DATA_BLOCK "DB7300_INTERLOCK_GENERAL"   // DB7300
{ S7_Optimized_Access := 'FALSE'; DB_Accessible_From_OPC_UA := 'FALSE' }
AUTHOR : ETXETAR
VERSION : 1.0
// stored: AutoNumber false, DBAccessibleFromOPCUA false, DBAccessibleFromWebserver true, IsOnlyStoredInLoadMemory false, IsWriteProtectedInAS false
   VAR RETAIN
      GENERAL_MACHINE : Struct
         FROM_CELL_TO_MACHINE_GENERAL : Struct
            MEAS_STA_START_CYCLE : Bool;   // CELL MEASURING STATION START CYCLE
            MEAS_STA_CALIB_CYCLE : Bool;   // CELL MEASURING STATION CALIBRATION CYCLE
            MEAS_STA_HOME_REQ : Bool;   // CELL MEASURING STATION HOME REQUEST
            MEAS_STA_FAULT : Bool;   // CELL MEASURING STATION FAULT
            MEAS_STA_RESET : Bool;   // CELL MEASURING STATION RESET
            MEAS_STA_ROBOT_OUT_OF_COLLISION : Bool;
            MEAS_STA_PART_LOADED : Bool;   // CELL MEASURING STATION PART LOADED
            MEAS_STA_PART_UNLOADED : Bool;   // CELL MEASURING STATION PART UNLOADED
            MEAS_STA_SEQ_RUNNING : Bool;   // CELL MEASURING STATION SEQUENCE RUNNING
            CELL_COOLING_DEGRADED_MODE : Bool;   // CELL COOLING DEGRADED MODE
            CELL_STARVED : Bool;   // CELL STARVED
            CELL_BLOCKED : Bool;   // CELL BLOCKED
            CELL_LOADING_ACTIVE : Bool;   // CELL LOADING ACTIVE
            CELL_CALIBRATION_CYCLE_REQUIRED : Bool;   // CELL CALIBRATION CYCLE REQUIRED
         END_STRUCT;
         FROM_ROBOT_TO_UNIT_1 : Struct
            HEARTBEAT : Bool;   // ROBOT HEARTBEAT
            EMERG_STOP_OK : Bool;   // ROBOT EMERGENCY STOP OK
            ROBOT_FAULT : Bool;   // ROBOT FAULT
            SAFETY_DOOR_CLSD_LOCKD : Bool;   // ROBOT SAFETY DOOR CLOSED AND LOCKED
            CELL_EMPTY : Bool;   // ROBOT CELL EMPTY
            IN_SEMIAUTO_MODE : Bool;   // ROBOT SEMIAUTO MODE SELECTED
            IN_MANUAL_MODE : Bool;   // ROBOT MANUAL MODE SELECTED
            IN_AUTO_MODE : Bool;   // ROBOT AUTO MODE SELECTED
            IN_AUTO_CYCLE_RUN : Bool;   // ROBOT CYCLE RUNNING IN AUTOMATIC MODE
            RUN_OUT_REQUEST : Bool;   // ROBOT MACHINE RUN OUT REQUEST
            RUN_OUT_COMPLETED : Bool;   // ROBOT RUN OUT COMPLETED
            SAFETY_DOOR_OPEN_REQ : Bool;   // ROBOT ANY CELL SAFETY DOOR OPEN REQUEST
            OK_TO_OPEN_SAFETY_GATES : Bool;   // ROBOT OK TO OPEN SAFETY GATES
            READY_TO_SERVICE : Bool;   // ROBOT READY TO SERVICE MACHINE
            OUT_OF_COLLISION_MACHINE : Bool;   // ROBOT OUT OF COLLISION MACHINE
            OUT_OF_COLLISION_FIXTURE : Bool;   // ROBOT OUT OF COLLISION FIXTURE
            PART_ENABLED : Bool;   // ROBOT PART ENABLED
            PART_FACE_R_TO_DELIVER : Bool;   // ROBOT PART FACE R TO DELIVER IMMEDIATELY
            PART_FACE_N_TO_DELIVER : Bool;   // ROBOT PART FACE N TO DELIVER IMMEDIATELY
            OUT_OF_PARTS_FACE_R_TO_DELIVER : Bool;   // ROBOT OUT OF PARTS FACE R IN CELL TO DELIVER
            OUT_OF_PARTS_FACE_N_TO_DELIVER : Bool;   // ROBOT OUT OF PARTS FACE N IN CELL TO DELIVER
            PART_LOADED : Bool;   // ROBOT PART LOADED
            PART_UNLOADED : Bool;   // ROBOT PART UNLOADED
            FIX_SKIP_REQ : Bool;   // ROBOT FIXTURE SKIP REQUEST
            PART_TYPE_CHANGE_REQ : Bool;   // ROBOT PART TYPE CHANGE REQUEST
            PART_TYPE : Byte;   // ROBOT PART TYPE
         END_STRUCT;
         FROM_ROBOT_TO_UNIT_2 : Struct
            HEARTBEAT : Bool;   // ROBOT HEARTBEAT
            EMERG_STOP_OK : Bool;   // ROBOT EMERGENCY STOP OK
            ROBOT_FAULT : Bool;   // ROBOT FAULT
            SAFETY_DOOR_CLSD_LOCKD : Bool;   // ROBOT SAFETY DOOR CLOSED AND LOCKED
            CELL_EMPTY : Bool;   // ROBOT CELL EMPTY
            IN_SEMIAUTO_MODE : Bool;   // ROBOT SEMIAUTO MODE SELECTED
            IN_MANUAL_MODE : Bool;   // ROBOT MANUAL MODE SELECTED
            IN_AUTO_MODE : Bool;   // ROBOT AUTO MODE SELECTED
            IN_AUTO_CYCLE_RUN : Bool;   // ROBOT CYCLE RUNNING IN AUTOMATIC MODE
            RUN_OUT_REQUEST : Bool;   // ROBOT MACHINE RUN OUT REQUEST
            RUN_OUT_COMPLETED : Bool;   // ROBOT RUN OUT COMPLETED
            SAFETY_DOOR_OPEN_REQ : Bool;   // ROBOT ANY CELL SAFETY DOOR OPEN REQUEST
            OK_TO_OPEN_SAFETY_GATES : Bool;   // ROBOT OK TO OPEN SAFETY GATES
            READY_TO_SERVICE : Bool;   // ROBOT READY TO SERVICE MACHINE
            OUT_OF_COLLISION_MACHINE : Bool;   // ROBOT OUT OF COLLISION MACHINE
            OUT_OF_COLLISION_FIXTURE : Bool;   // ROBOT OUT OF COLLISION FIXTURE
            PART_ENABLED : Bool;   // ROBOT PART ENABLED
            PART_FACE_R_TO_DELIVER : Bool;   // ROBOT PART FACE R TO DELIVER IMMEDIATELY
            PART_FACE_N_TO_DELIVER : Bool;   // ROBOT PART FACE N TO DELIVER IMMEDIATELY
            OUT_OF_PARTS_FACE_R_TO_DELIVER : Bool;   // ROBOT OUT OF PARTS FACE R IN CELL TO DELIVER
            OUT_OF_PARTS_FACE_N_TO_DELIVER : Bool;   // ROBOT OUT OF PARTS FACE N IN CELL TO DELIVER
            PART_LOADED : Bool;   // ROBOT PART LOADED
            PART_UNLOADED : Bool;   // ROBOT PART UNLOADED
            FIX_SKIP_REQ : Bool;   // ROBOT FIXTURE SKIP REQUEST
            PART_TYPE_CHANGE_REQ : Bool;   // ROBOT PART TYPE CHANGE REQUEST
            PART_TYPE : Byte;   // ROBOT PART TYPE
         END_STRUCT;
      END_STRUCT;
      POWDER_PLC : Struct
         GENERAL : Struct
            LIFE_BIT : Bool;   // LIFE BIT
            SELECTED_ARGON_GAS : Bool;   // SELECTED ARGON GAS
            SELECTED_NITROGEN_GAS : Bool;   // SELECTED NITROGEN GAS
            SELECTED_IMPERIAL_SYSTEM : Bool;   // SELECTED IMPERIAL SYSTEM
            SELECTED_METRIC_SYSTEM : Bool;   // SELECTED METRIC SYSTEM
            POWDER_PLC_AUTO_MODE : Bool;   // POWDER PLC IN AUTO MODE
            POWDER_PLC_MAN_MODE : Bool;   // POWDER PLC IN MANUAL MODE
         END_STRUCT;
         FROM_POWDER_TO_UNIT_1 : Struct
            POWDER_UNIT_1_READY_TO_RUN : Bool;   // POWDER UNIT 1 READY TO RUN
            POWDER_UNIT_1_STOPPED : Bool;   // POWDER UNIT 1 STOPPED
            SWITCHED_ON_POWDER_UNIT_1 : Bool;   // SWITCHED ON POWDER UNIT 1
            SWITCHED_OFF_POWDER_UNIT_1 : Bool;   // SWITCHED OFF POWDER UNIT 1
            SWITCHED_ON_TEMPERATURE_JACKET_UNIT_1 : Bool;   // SWITCHED ON TEMPERATURE JACKET UNIT 1
            SWITCHED_OFF_TEMPERATURE_JACKET_UNIT_1 : Bool;   // SWITCHED OFF TEMPERATURE JACKET UNIT 1
            U1_PF_1_LINE_1_LOW_POWDER : Bool;   // UNIT 1 POWDER FEEDER 1 LINE 1 LOW POWDER LEVEL
            U1_PF_1_LINE_2_LOW_POWDER : Bool;   // UNIT 1 POWDER FEEDER 1 LINE 2 LOW POWDER LEVEL
            POWDER_UNIT_1_ALARM : Bool;   // POWDER UNIT 1 ALARM
            UNIT_1_POWDER_FEEDER_1_CARRIER_GAS_ACTUAL_LINE_1 : Real;   // UNIT 1 POWDER FEEDER 1 CARRIER GAS ACTUAL LINE 1
            UNIT_1_POWDER_FEEDER_1_DISK_SPEED_ACTUAL_LINE_1 : Real;   // UNIT 1 POWDER FEEDER 1 DISK SPEED ACTUAL LINE 1
            UNIT_1_POWDER_FEEDER_1_STIRRER_SPEED_ACTUAL_LINE_1 : Real;   // UNIT 1 POWDER FEEDER 1 STIRRER SPEED ACTUAL LINE 1
            UNIT_1_POWDER_FEEDER_1_HOPPER_TEMPERATURE_ACTUAL_LINE_1 : Real;   // UNIT 1 POWDER FEEDER 1 HOPPER TEMPERATURE ACTUAL LINE 1
            UNIT_1_POWDER_FEEDER_1_CARRIER_GAS_ACTUAL_LINE_2 : Real;   // UNIT 1 POWDER FEEDER 1 CARRIER GAS ACTUAL LINE 2
            UNIT_1_POWDER_FEEDER_1_DISK_SPEED_ACTUAL_LINE_2 : Real;   // UNIT 1 POWDER FEEDER 1 DISK SPEED ACTUAL LINE 2
            UNIT_1_POWDER_FEEDER_1_STIRRER_SPEED_ACTUAL_LINE_2 : Real;   // UNIT 1 POWDER FEEDER 1 STIRRER SPEED ACTUAL LINE 2
            UNIT_1_POWDER_FEEDER_1_HOPPER_TEMPERATURE_ACTUAL_LINE_2 : Real;   // UNIT 1 POWDER FEEDER 1 HOPPER TEMPERATURE ACTUAL LINE 2
         END_STRUCT;
         FROM_POWDER_TO_UNIT_2 : Struct
            POWDER_UNIT_2_READY_TO_RUN : Bool;   // POWDER UNIT 2 READY TO RUN
            POWDER_UNIT_2_STOPPED : Bool;   // POWDER UNIT 2 STOPPED
            SWITCHED_ON_POWDER_UNIT_2 : Bool;   // SWITCHED ON POWDER UNIT 2
            SWITCHED_OFF_POWDER_UNIT_2 : Bool;   // SWITCHED OFF POWDER UNIT 2
            SWITCHED__ON_TEMPERATURE_JACKET_UNIT_2 : Bool;   // SWITCHED ON TEMPERATURE JACKET UNIT 2
            SWITCHED_OFF_TEMPERATURE_JACKET_UNIT_2 : Bool;   // SWITCHED OFF TEMPERATURE JACKET UNIT 2
            U2_PF_1_LINE_1_LOW_POWDER : Bool;   // UNIT 2 POWDER FEEDER 1 LINE 1 LOW POWDER LEVEL
            U2_PF_1_LINE_2_LOW_POWDER : Bool;   // UNIT 2 POWDER FEEDER 1 LINE 2 LOW POWDER LEVEL
            U2_PF_2_LINE_2_LOW_POWDER : Bool;   // UNIT 2 POWDER FEEDER 2 LINE 2 LOW POWDER LEVEL
            POWDER_UNIT_2_ALARM : Bool;   // POWDER UNIT 2 ALARM
            UNIT_2_POWDER_FEEDER_1_CARRIER_GAS_ACTUAL_LINE_1 : Real;   // UNIT 2 POWDER FEEDER 1 CARRIER GAS ACTUAL LINE 1
            UNIT_2_POWDER_FEEDER_1_CARRIER_GAS_ACTUAL_LINE_2 : Real;   // UNIT 2 POWDER FEEDER 1 CARRIER GAS ACTUAL LINE 2
            UNIT_2_POWDER_FEEDER_1_DISK_SPEED_ACTUAL_LINE_1 : Real;   // UNIT 2 POWDER FEEDER 1 DISK SPEED ACTUAL LINE 1
            UNIT_2_POWDER_FEEDER_1_DISK_SPEED_ACTUAL_LINE_2 : Real;   // UNIT 2 POWDER FEEDER 1 DISK SPEED ACTUAL LINE 2
            UNIT_2_POWDER_FEEDER_1_STIRRER_SPEED_ACTUAL_LINE_1 : Real;   // UNIT 2 POWDER FEEDER 1 STIRRER SPEED ACTUAL LINE 1
            UNIT_2_POWDER_FEEDER_1_STIRRER_SPEED_ACTUAL_LINE_2 : Real;   // UNIT 2 POWDER FEEDER 1 STIRRER SPEED ACTUAL LINE 2
            UNIT_2_POWDER_FEEDER_1_HOPPER_TEMPERATURE_ACTUAL_LINE_1 : Real;   // UNIT 2 POWDER FEEDER 1 HOPPER TEMPERATURE ACTUAL LINE 1
            UNIT_2_POWDER_FEEDER_1_HOPPER_TEMPERATURE_ACTUAL_LINE_2 : Real;   // UNIT 2 POWDER FEEDER 1 HOPPER TEMPERATURE ACTUAL LINE 2
            UNIT_2_POWDER_FEEDER_2_CARRIER_GAS_ACTUAL_LINE_1 : Real;   // UNIT 2 POWDER FEEDER 2 CARRIER GAS ACTUAL LINE 1
            UNIT_2_POWDER_FEEDER_2_CARRIER_GAS_ACTUAL_LINE_2 : Real;   // UNIT 2 POWDER FEEDER 2 CARRIER GAS ACTUAL LINE 2
            UNIT_2_POWDER_FEEDER_2_DISK_SPEED_ACTUAL_LINE_1 : Real;   // UNIT 2 POWDER FEEDER 2 DISK SPEED ACTUAL LINE 1
            UNIT_2_POWDER_FEEDER_2_STIRRER_SPEED_ACTUAL_LINE_1 : Real;   // UNIT 2 POWDER FEEDER 2 STIRRER SPEED ACTUAL LINE 1
            UNIT_2_POWDER_FEEDER_2_DISK_SPEED_ACTUAL_LINE_2 : Real;   // UNIT 2 POWDER FEEDER 2 DISK SPEED ACTUAL LINE 2
            UNIT_2_POWDER_FEEDER_2_STIRRER_SPEED_ACTUAL_LINE_2 : Real;   // UNIT 2 POWDER FEEDER 2 STIRRER SPEED ACTUAL LINE 2
            UNIT_2_POWDER_FEEDER_2_HOPPER_TEMPERATURE_ACTUAL_LINE_1 : Real;   // UNIT 2 POWDER FEEDER 2 HOPPER TEMPERATURE ACTUAL LINE 1
            UNIT_2_POWDER_FEEDER_2_HOPPER_TEMPERATURE_ACTUAL_LINE_2 : Real;   // UNIT 2 POWDER FEEDER 2 HOPPER TEMPERATURE ACTUAL LINE 2
         END_STRUCT;
      END_STRUCT;
      LOAD_UNLOAD : Struct
         UNIT_1 : "LOAD_UNLOAD_ETXETAR_ROBOT_CELL";
         UNIT_2 : "LOAD_UNLOAD_ETXETAR_ROBOT_CELL";
         UNIT_3 : "LOAD_UNLOAD_ETXETAR_ROBOT_CELL";
      END_STRUCT;
      AUX_SIGNALS_INTERFACE : Struct
         GENERAL : Struct
            "MEASURING STATION FAULT" : Bool;   // CELL MEASURING STATION FAULT
            "DEGRADED MODE FAULT" : Bool;   // CELL COOLING DEGRADED MODE FAULT
            TIMER_MEASURING_IN_PRCS : TOF_TIME;   // TIMER MEASURING IN PROCESS
            TIMER_MEASURING_DONE : TOF_TIME;   // TIMER MEASURING DONE
         END_STRUCT;
         UNIT_1 : Struct
            LIFE_BIT_FAULT : Bool;   // HEARTBEAT COMMUNICATION ALARM
            EMERGENCY_STOP_ACTIVE : Bool;   // EMERGENCY STOP ACTIVE ALARM
            ROBOT_FAULT_INSIDE_OF_MACHINE : Bool;   // ROBOT FAULT ALARM INSIDE OF MACHINE
            ROBOT_FAULT_OUTSIDE_OF_MACHINE : Bool;   // ROBOT FAULT ALARM OUTSIDE OF MACHINE
            FACE_R_LOAD_REQ_AUX : Bool;   // FACE R LOAD REQUEST AUX
            FACE_N_LOAD_REQ_AUX : Bool;   // FACE N LOAD REQUEST AUX
            "LIFE SING COUNTER" : CTU_INT;
         END_STRUCT;
         UNIT_2 : Struct
            LIFE_BIT_FAULT : Bool;   // HEARTBEAT COMMUNICATION ALARM
            EMERGENCY_STOP_ACTIVE : Bool;   // EMERGENCY STOP ACTIVE ALARM
            ROBOT_FAULT_INSIDE_OF_MACHINE : Bool;   // ROBOT FAULT ALARM INSIDE OF MACHINE
            ROBOT_FAULT_OUTSIDE_OF_MACHINE : Bool;   // ROBOT FAULT ALARM OUTSIDE OF MACHINE
            FACE_R_LOAD_REQ_AUX : Bool;   // FACE R LOAD REQUEST AUX
            FACE_N_LOAD_REQ_AUX : Bool;   // FACE N LOAD REQUEST AUX
            "LIFE SING COUNTER" : CTU_INT;
         END_STRUCT;
         POWDER_PLC : Struct
            LIFE_BIT_FAULT : Bool;   // HEARTBEAT COMMUNICATION ALARM
            "LIFE SING COUNTER" : CTU_INT;
         END_STRUCT;
         AUX_0 : Bool;   // AUXILIARY 0
         AUX_1 : Bool;   // AUXILIARY 1
         AUX_2 : Bool;   // AUXILIARY 2
         AUX_3 : Bool;   // AUXILIARY 3
         AUX_4 : Bool;   // AUXILIARY 4
         AUX_5 : Bool;   // AUXILIARY 5
         AUX_6 : Bool;   // AUXILIARY 6
         AUX_7 : Bool;   // AUXILIARY 7
         AUX_8 : Bool;   // AUXILIARY 8
         AUX_9 : Bool;   // AUXILIARY 9
         AUX_10 : Bool;   // AUXILIARY 10
         AUX_11 : Bool;   // AUXILIARY 11
         AUX_12 : Bool;   // AUXILIARY 12
         AUX_13 : Bool;   // AUXILIARY 13
         AUX_14 : Bool;   // AUXILIARY 14
         AUX_15 : Bool;   // AUXILIARY 15
         TIMER_IS_SEOC_ROBOT_FAULT_UNIT_1 : TON_TIME;   // TIMER IS SEOC ROBOT FAULT UNIT 1
         TIMER_IS_SEOC_ROBOT_FAULT_UNIT_2 : TON_TIME;   // TIMER IS SEOC ROBOT FAULT UNIT 2
         TIMER_SEOC_ROBOT_FAULT_UNIT_1 : TON_TIME;   // TIMER SEOC ROBOT FAULT UNIT 1
         TIMER_SEOC_ROBOT_FAULT_UNIT_2 : TON_TIME;   // TIMER SEOC ROBOT FAULT UNIT 2
      END_STRUCT;
      PART_A : Struct
         UNIT_1 : "PART_STATUS_CLADDING";
         UNIT_2 : "PART_STATUS_CLADDING";
         UNIT_3 : "PART_STATUS_CLADDING";
      END_STRUCT;
   END_VAR
BEGIN
   AUX_SIGNALS_INTERFACE.GENERAL.TIMER_MEASURING_IN_PRCS.PT := T#3s;
   AUX_SIGNALS_INTERFACE.GENERAL.TIMER_MEASURING_DONE.PT := T#3s;
   AUX_SIGNALS_INTERFACE.TIMER_IS_SEOC_ROBOT_FAULT_UNIT_1.PT := T#2M;
   AUX_SIGNALS_INTERFACE.TIMER_IS_SEOC_ROBOT_FAULT_UNIT_2.PT := T#2M;
   AUX_SIGNALS_INTERFACE.TIMER_SEOC_ROBOT_FAULT_UNIT_1.PT := T#2M;
   AUX_SIGNALS_INTERFACE.TIMER_SEOC_ROBOT_FAULT_UNIT_2.PT := T#2M;
END_DATA_BLOCK

DATA_BLOCK "DB7400_QUALITY"   // DB7400
{ S7_Optimized_Access := 'FALSE'; DB_Accessible_From_OPC_UA := 'FALSE' }
AUTHOR : ETXETAR
VERSION : 1.0
// stored: AutoNumber false, DBAccessibleFromOPCUA false, DBAccessibleFromWebserver true, IsOnlyStoredInLoadMemory false, IsWriteProtectedInAS false
   VAR RETAIN
      OPTIONS : Struct   // OPTIONS
         QC_STOP_END_OF_CYCLE : Bool;   // QC STOP END OF CYCLE
         SP11_WORKS_TWO_PARTS : Bool;   // SP11 WORKS TWO PARTS
         SP12_WORKS_TWO_PARTS : Bool;   // SP12 WORKS TWO PARTS
         SP21_WORKS_TWO_PARTS : Bool;   // SP21 WORKS TWO PARTS
         SP22_WORKS_TWO_PARTS : Bool;   // SP22 WORKS TWO PARTS
         FIRST_SCAN : Bool;   // FIRST SCAN
         CYCLE_INTERRUPTED : Bool;   // CYCLE INTERRUPTED
         ANY_TOOL_NEW : Bool;   // ANY TOOL NEW
         BROKEN_TOOL : Bool;   // BROKEN TOOL
         ALL_BROKEN_TOOL : Bool;   // ALL BROKEN TOOL IF ONE TOOL IS BROKEN ALL PARTS ARE MARKED
         ONE_COUNTER : Bool;   // ONE COUNTER
         COUNTER_PER_PART : Bool;   // COUNTER PER PART
         CMM_QUALITY_CHECK : Bool;   // CMM QUALITY CHECK
         SURFACE_QUALITY_CHECK : Bool;   // SURFACE QUALITY CHECK
      END_STRUCT;
      PART_CONTROL : Struct   // PART CONTROL
         HMI_QUALITY_HALF_PART : Bool;   // HMI QUALITY HALF PART
         HMI_QUALITY_FULL_PART : Bool;   // HMI QUALITY FULL PART
         HMI_QUALITY_CANCEL : Bool;   // HMI QUALITY CANCEL
         HMI_QUALITY_NOK : Bool;   // HMI QUALITY NOK
         HMI_QUALITY_OK : Bool;   // HMI QUALITY OK
         HALF_QUALITY_PART_SELECTED : Bool;   // HALF QUALITY PART SELECTED
         FULL_QUALITY_PART_SELECTED : Bool;   // FULL QUALITY PART SELECTED
         PART_QUALITY_ON_DEMAND : Bool;   // PART QUALITY ON DEMAND
         QUALITY_AUX_WARNING : Bool;   // QUALITY AUX WARNING
         QUALITY_AUX_FAULT : Bool;   // QUALITY AUX FAULT
         QUALITY_PART : Bool;   // QUALITY PART
         FIXTURE_2_QUALITY : Bool;   // FIXTURE 2 QUALITY
         U01_FIXTURE_1_PART_P : Bool;   // UNIT 01 FIXTURE 1 PART A PULSE
         U01_FIXTURE_2_PART_P : Bool;   // UNIT 01 FIXTURE 2 PART A PULSE
         U01_FIXTURE_3_PART_P : Bool;   // UNIT 01 FIXTURE 3 PART A PULSE
         U01_FIXTURE_4_PART_P : Bool;   // UNIT 01 FIXTURE 4 PART A PULSE
         U02_FIXTURE_1_PART_P : Bool;   // UNIT 02 FIXTURE 1 PART A PULSE
         U02_FIXTURE_2_PART_P : Bool;   // UNIT 02 FIXTURE 2 PART A PULSE
         U02_FIXTURE_3_PART_P : Bool;   // UNIT 02 FIXTURE 3 PART A PULSE
         U02_FIXTURE_4_PART_P : Bool;   // UNIT 02 FIXTURE 4 PART A PULSE
         U01_FIXTURE_1_PART_DEMAND : Bool;   // UNIT 01 FIXTURE 1 PART A DEMAND
         U01_FIXTURE_2_PART_DEMAND : Bool;   // UNIT 01 FIXTURE 2 PART A DEMAND
         U01_FIXTURE_3_PART_DEMAND : Bool;   // UNIT 01 FIXTURE 3 PART A DEMAND
         U01_FIXTURE_4_PART_DEMAND : Bool;   // UNIT 01 FIXTURE 4 PART A DEMAND
         U02_FIXTURE_1_PART_DEMAND : Bool;   // UNIT 02 FIXTURE 1 PART A DEMAND
         U02_FIXTURE_2_PART_DEMAND : Bool;   // UNIT 02 FIXTURE 2 PART A DEMAND
         U02_FIXTURE_3_PART_DEMAND : Bool;   // UNIT 02 FIXTURE 3 PART A DEMAND
         U02_FIXTURE_4_PART_DEMAND : Bool;   // UNIT 02 FIXTURE 4 PART A DEMAND
         PART_NOK : Bool;   // PART QUALITY DEMAND NOK ALARM
      END_STRUCT;
      PART_TYPE : Struct   // PART TYPE
         PART_TYPE_CHANGE_AUX : Bool;   // PART TYPE CHANGE AUXILIARY
         FIXTURE_1_PART_TYPE_CHANGE : Bool;   // FIXTURE 1 PART TYPE CHANGE
         FIXTURE_2_PART_TYPE_CHANGE : Bool;   // FIXTURE 2 PART TYPE CHANGE
         FIXTURE_3_PART_TYPE_CHANGE : Bool;   // FIXTURE 3 PART TYPE CHANGE
         FIXTURE_4_PART_TYPE_CHANGE : Bool;   // FIXTURE 4 PART TYPE CHANGE
         QUALITY_PART_TYPE_CHANGE : Bool;   // QUALITY AFTER PART TYPE CHANGE
         QUALITY_PART_NOK : Bool;   // QUALITY PART AFTER PART TYPE CHANGE NOK ALARM
      END_STRUCT;
      FIRST_CYCLE : Struct   // FIRST CYCLE
         FIRST_SCAN_AUX : Bool;   // FIRST SCAN AUXILIARY
         QUALITY_FIRST_CYCLE : Bool;   // QUALITY FIRST CYCLE
         FIXTURE_2_FIRST_CYCLE : Bool;   // FIXTURE 2 FIRST CYCLE
         FIXTURE_1_PART_A : Bool;   // FIXTURE 1 PART A FIRST CYCLE
         FIXTURE_1_PART_A_NOK : Bool;   // FIXTURE 1 PART A FIRST CYCLE NOK ALARM
      END_STRUCT;
      CYCLE_INTERRUPTED : Struct   // CYCLE INTERRUPTED
         CYCLE_INTERRUPTED_AUX : Bool;   // CYCLE INTERRUPTED AUXILIARY
         CYCLE_INTERRUPTED_AUX_P : Bool;   // CYCLE INTERRUPTED AUXILIARY PULSE
         FIXTURE_1_CYCLE_INTERRUPTED : Bool;   // FIXTURE 1 CYCLE INTERRUPTED
         FIXTURE_2_CYCLE_INTERRUPTED : Bool;   // FIXTURE 2 CYCLE INTERRUPTED
         FIXTURE_1_PART_A : Bool;   // FIXTURE 1 PART A CYCLE INTERRUPTED
         FIXTURE_1_PART_B : Bool;   // FIXTURE 1 PART B CYCLE INTERRUPTED
         FIXTURE_1_PART_C : Bool;   // FIXTURE 1 PART C CYCLE INTERRUPTED
         FIXTURE_1_PART_D : Bool;   // FIXTURE 1 PART D CYCLE INTERRUPTED
         FIXTURE_2_PART_A : Bool;   // FIXTURE 2 PART A CYCLE INTERRUPTED
         FIXTURE_2_PART_B : Bool;   // FIXTURE 2 PART B CYCLE INTERRUPTED
         FIXTURE_2_PART_C : Bool;   // FIXTURE 2 PART C CYCLE INTERRUPTED
         FIXTURE_2_PART_D : Bool;   // FIXTURE 2 PART D CYCLE INTERRUPTED
         FIXTURE_1_PART_A_NOK : Bool;   // FIXTURE 1 PART A CYCLE INTERRUPTED NOK ALARM
         FIXTURE_1_PART_B_NOK : Bool;   // FIXTURE 1 PART B CYCLE INTERRUPTED NOK ALARM
         FIXTURE_1_PART_C_NOK : Bool;   // FIXTURE 1 PART C CYCLE INTERRUPTED NOK ALARM
         FIXTURE_1_PART_D_NOK : Bool;   // FIXTURE 1 PART D CYCLE INTERRUPTED NOK ALARM
         FIXTURE_2_PART_A_NOK : Bool;   // FIXTURE 2 PART A CYCLE INTERRUPTED NOK ALARM
         FIXTURE_2_PART_B_NOK : Bool;   // FIXTURE 2 PART B CYCLE INTERRUPTED NOK ALARM
         FIXTURE_2_PART_C_NOK : Bool;   // FIXTURE 2 PART C CYCLE INTERRUPTED NOK ALARM
         FIXTURE_2_PART_D_NOK : Bool;   // FIXTURE 2 PART D CYCLE INTERRUPTED NOK ALARM
         S_PECT_01 : TP_TIME;   // S PECT 01
      END_STRUCT;
      PART_COUNTER : Struct   // PART COUNTER
         PART_COUNTER_REACHED_AUX : Bool;   // PART COUNTR REACHED AUXILIARY
         PARTS_COUNTER_AUX_P : Bool;   // PARTS COUNTER AUX PULSE
         QUALITY_PART_COUNTER_REACHED : Bool;   // QUALITY AFTER PART COUNTER REACHED
         QUALITY_PART_NOK : Bool;   // QUALITY PART AFTER PART COUNTER REACHED ALARM
      END_STRUCT;
      QUALITY_AUX_DATA : Struct   // QUALITY AUXILIARY DATA
         PARTS_COUNTER : Int := 0;   // PARTS COUNTER
         QUALITY_AFTER_PARTS : Int;   // PARTS BEFORE CHECK QUALITY
      END_STRUCT;
   END_VAR
BEGIN
END_DATA_BLOCK

DATA_BLOCK "DB8000_PART_STATUS"   // DB8000
{ S7_Optimized_Access := 'FALSE'; DB_Accessible_From_OPC_UA := 'FALSE' }
AUTHOR : ETXETAR
VERSION : 1.0
// stored: AutoNumber false, DBAccessibleFromOPCUA false, DBAccessibleFromWebserver true, IsOnlyStoredInLoadMemory false, IsWriteProtectedInAS false
   VAR RETAIN
      HMI : Struct
         ONE_PART_LOADED_FOR_MACH : Bool;   // ONE PART LOADED FOR MACH
         UNIT_01_PART_PRESENT : Bool;   // HMI UNIT 01 PART PRESENT BUTTON
         UNIT_01_REMOVE_PART : Bool;   // HMI UNIT 01 REMOVE PART BUTTON
         UNIT_01_GOOD_PART : Bool;   // HMI UNIT 01 GOOD PART NOT MACHINED BUTTON
         UNIT_01_REJECT_PART : Bool;   // HMI UNIT 01 NOT OK PART BUTTON
         UNIT_01_MASTER_PART : Bool;   // HMI UNIT 01 SET MASTER PART
         UNIT_02_PART_PRESENT : Bool;   // HMI UNIT 02 PART PRESENT BUTTON
         UNIT_02_REMOVE_PART : Bool;   // HMI UNIT 02 REMOVE PART BUTTON
         UNIT_02_GOOD_PART : Bool;   // HMI UNIT 02 GOOD PART NOT MACHINED BUTTON
         UNIT_02_REJECT_PART : Bool;   // HMI UNIT 02 NOT OK PART BUTTON
         UNIT_02_MASTER_PART : Bool;   // HMI UNIT 02 SET MASTER PART
         UNIT_03_PART_PRESENT : Bool;   // HMI UNIT 03 PART PRESENT BUTTON
         UNIT_03_REMOVE_PART : Bool;   // HMI UNIT 03 REMOVE PART BUTTON
         UNIT_03_GOOD_PART : Bool;   // HMI UNIT 03 GOOD PART NOT MACHINED BUTTON
         UNIT_03_REJECT_PART : Bool;   // HMI UNIT 03 NOT OK PART BUTTON
         UNIT_03_MASTER_PART : Bool;   // HMI UNIT 03 SET MASTER PART
         PART_STATUS_FIXTURES_LIST : Int := 1;   // HMI PART STATUS FIXTURES LIST
         PART_STATUS_PART_TYPE_LIST : Int := 1;   // HMI PART STATUS PART TYPE LIST
         PART_STATUS_PART_STATUS_LIST : Int := 1;   // HMI PART STATUS PROCESS PART STATUS LIST
         PART_NUMBER_LIST : Int;   // PART TYPE LIST AUX
      END_STRUCT;
      UNIT_1 : Struct
         FIXTURE_1 : Struct
            PART_A { S7_SetPoint := 'True'} : "PART_STATUS_CLADDING";
         END_STRUCT;
         FIXTURE_2 : Struct
            PART_A { S7_SetPoint := 'True'} : "PART_STATUS_CLADDING";
         END_STRUCT;
         FIXTURE_3 : Struct
            PART_A { S7_SetPoint := 'True'} : "PART_STATUS_CLADDING";
         END_STRUCT;
         FIXTURE_4 : Struct
            PART_A { S7_SetPoint := 'True'} : "PART_STATUS_CLADDING";
         END_STRUCT;
         STATION_1 : Struct
            PART_A { S7_SetPoint := 'True'} : "PART_STATUS_CLADDING";
         END_STRUCT;
         STATION_2 : Struct
            PART_A { S7_SetPoint := 'True'} : "PART_STATUS_CLADDING";
         END_STRUCT;
         STATION_3 : Struct
            PART_A { S7_SetPoint := 'True'} : "PART_STATUS_CLADDING";
         END_STRUCT;
         STATION_4 : Struct
            PART_A { S7_SetPoint := 'True'} : "PART_STATUS_CLADDING";
         END_STRUCT;
      END_STRUCT;
      UNIT_2 : Struct
         FIXTURE_1 : Struct
            PART_A { S7_SetPoint := 'True'} : "PART_STATUS_CLADDING";
         END_STRUCT;
         FIXTURE_2 : Struct
            PART_A { S7_SetPoint := 'True'} : "PART_STATUS_CLADDING";
         END_STRUCT;
         FIXTURE_3 : Struct
            PART_A { S7_SetPoint := 'True'} : "PART_STATUS_CLADDING";
         END_STRUCT;
         FIXTURE_4 : Struct
            PART_A { S7_SetPoint := 'True'} : "PART_STATUS_CLADDING";
         END_STRUCT;
         STATION_1 : Struct
            PART_A { S7_SetPoint := 'True'} : "PART_STATUS_CLADDING";
         END_STRUCT;
         STATION_2 : Struct
            PART_A { S7_SetPoint := 'True'} : "PART_STATUS_CLADDING";
         END_STRUCT;
         STATION_3 : Struct
            PART_A { S7_SetPoint := 'True'} : "PART_STATUS_CLADDING";
         END_STRUCT;
         STATION_4 : Struct
            PART_A { S7_SetPoint := 'True'} : "PART_STATUS_CLADDING";
         END_STRUCT;
      END_STRUCT;
      UNIT_3 : Struct
         FIXTURE_1 : Struct
            PART_A { S7_SetPoint := 'True'} : "PART_STATUS_CLADDING";
         END_STRUCT;
      END_STRUCT;
      PULSE_1 : Bool;   // PULSE 1
      PULSE_2 : Bool;   // PULSE 2
      PULSE_3 : Bool;   // PULSE 3
      PULSE_4 : Bool;   // PULSE 4
      PULSE_5 : Bool;   // PULSE 5
      PULSE_6 : Bool;   // PULSE 6
      PULSE_7 : Bool;   // PULSE 7
      PULSE_8 : Bool;   // PULSE 8
      PULSE_9 : Bool;   // PULSE 9
      PULSE_10 : Bool;   // PULSE 10
      PULSE_11 : Bool;   // PULSE 11
      PULSE_12 : Bool;   // PULSE 12
      PULSE_13 : Bool;   // PULSE 13
      PULSE_14 : Bool;   // PULSE 14
      PULSE_15 : Bool;   // PULSE 15
      PULSE_16 : Bool;   // PULSE 16
      PULSE_17 : Bool;   // PULSE 17
      PULSE_18 : Bool;   // PULSE 18
      PULSE_19 : Bool;   // PULSE 19
      PULSE_20 : Bool;   // PULSE 20
      PULSE_21 : Bool;   // PULSE 21
      PULSE_22 : Bool;   // PULSE 22
      PULSE_23 : Bool;   // PULSE 23
      PULSE_24 : Bool;   // PULSE 24
   END_VAR
BEGIN
END_DATA_BLOCK

DATA_BLOCK "DB8001_UNIT_1_PART_STATUS_HMI"   // DB8001
{ S7_Optimized_Access := 'FALSE'; DB_Accessible_From_OPC_UA := 'FALSE' }
VERSION : 0.1
// stored: AutoNumber false, DBAccessibleFromOPCUA false, DBAccessibleFromWebserver true, IsOnlyStoredInLoadMemory false, IsWriteProtectedInAS false
   VAR
      Int_PART_TYPE : Array[0..63] of Char;
      WChar_PART_TYPE : Array[0..63] of WChar;
   END_VAR
BEGIN
END_DATA_BLOCK

DATA_BLOCK "DB8002_UNIT_02_PART_STATUS_HMI"   // DB8002
{ S7_Optimized_Access := 'FALSE'; DB_Accessible_From_OPC_UA := 'FALSE' }
VERSION : 0.1
// stored: AutoNumber false, DBAccessibleFromOPCUA false, DBAccessibleFromWebserver true, IsOnlyStoredInLoadMemory false, IsWriteProtectedInAS false
   VAR
      Int_PART_TYPE : Array[0..63] of Char;
      WChar_PART_TYPE : Array[0..63] of WChar;
   END_VAR
BEGIN
END_DATA_BLOCK

DATA_BLOCK "DB8100_MANUAL_LOADING_PART_STATUS"   // DB8100
{ S7_Optimized_Access := 'FALSE'; DB_Accessible_From_OPC_UA := 'FALSE' }
VERSION : 0.1
// stored: AutoNumber false, DBAccessibleFromOPCUA false, DBAccessibleFromWebserver true, IsOnlyStoredInLoadMemory false, IsWriteProtectedInAS false
   VAR
      UNIT_01_DELETE_PART_HMI_BUTTON : Bool;   // DELETE PART FROM FIXTURE IN UNIT 01 STATION 1 HMI BUTTON
      UNIT_01_ADD_PART_HMI_BUTTON : Bool;   // ADD PART TO FIXTURE IN UNIT 01 STATION 1 HMI BUTTON
      UNIT_01_SKIP_LOADING_FIX_STA_1_HMI_BUTTON : Bool;   // UNIT 01 SKIP LOADING FIXTURE IN STATION 1 HMI BUTTON
      UNIT_01_NO_FACE_R_PARTS_TO_DELIVER : Bool;   // NO FACE R PARTS TO DELIVER UNIT 01
      UNIT_01_NO_FACE_N_PARTS_TO_DELIVER : Bool;   // NO FACE N PARTS TO DELIVER UNIT 01
      UNIT_01_SPARE_3 : Bool;
      UNIT_01_SPARE_4 : Bool;
      UNIT_01_SPARE_5 : Bool;
      UNIT_02_DELETE_PART_HMI_BUTTON : Bool;   // DELETE PART FROM FIXTURE IN UNIT 02 STATION 1 HMI BUTTON
      UNIT_02_ADD_PART_HMI_BUTTON : Bool;   // ADD PART TO FIXTURE IN UNIT 02 STATION 1 HMI BUTTON
      UNIT_02_SKIP_LOADING_FIX_STA_1_HMI_BUTTON : Bool;   // UNIT 02 SKIP LOADING FIXTURE IN STATION 1 HMI BUTTON
      UNIT_02_NO_FACE_R_PARTS_TO_DELIVER : Bool;   // NO FACE R PARTS TO DELIVER UNIT 02
      UNIT_02_NO_FACE_N_PARTS_TO_DELIVER : Bool;   // NO FACE N PARTS TO DELIVER UNIT 02
      UNIT_02_SPARE_3 : Bool;
      UNIT_02_SPARE_4 : Bool;
      UNIT_02_SPARE_5 : Bool;
      UNIT_03_DELETE_PART_HMI_BUTTON : Bool;   // DELETE PART FROM FIXTURE IN UNIT 03 STATION 1 HMI BUTTON
      UNIT_03_ADD_PART_HMI_BUTTON : Bool;   // ADD PART TO FIXTURE IN UNIT 03 STATION 1 HMI BUTTON
      UNIT_03_SPARE_1 : Bool;
      UNIT_03_SPARE_2 : Bool;
      UNIT_03_SPARE_3 : Bool;
      UNIT_03_SPARE_4 : Bool;
      UNIT_03_SPARE_5 : Bool;
      UNIT_03_SPARE_6 : Bool;
   END_VAR
BEGIN
END_DATA_BLOCK

DATA_BLOCK "DB8101_MANUAL_LOADING_PART_STATUS_MANAGEMENT"   // DB8101
{ S7_Optimized_Access := 'FALSE'; DB_Accessible_From_OPC_UA := 'FALSE' }
VERSION : 0.1
// stored: AutoNumber false, DBAccessibleFromOPCUA false, DBAccessibleFromWebserver true, IsOnlyStoredInLoadMemory false, IsWriteProtectedInAS false
   VAR
      UNIT_01_INTERMEDIATE : "PART_STATUS_CLADDING";
      UNIT_01_UNIT_02_INTERMEDIATE : "PART_STATUS_CLADDING";
      UNIT_02_INTERMEDIATE : "PART_STATUS_CLADDING";
   END_VAR
BEGIN
END_DATA_BLOCK

ORGANIZATION_BLOCK "OB1_CYCLE"   // OB1, LAD, ProgramCycle
TITLE = "Main Program Sweep (Cycle)"
{ S7_Optimized_Access := 'FALSE' }
AUTHOR : ETXETAR
VERSION : 1.0
// stored: AutoNumber false, IsIECCheckEnabled false, SetENOAutomatically false
   VAR_TEMP
      OB1_SCAN : Byte;   // 1 (Cold restart scan 1 of OB 1), 3 (Scan 2-n of OB 1)
      OB1_PRIORITY : Int;   // Priority of OB Execution
      OB1_MIN_CYCLE : DInt;   // Minimum cycle time of OB1 (milliseconds)
      OB1_MAX_CYCLE : DInt;   // Maximum cycle time of OB1 (milliseconds)
      PART_TYPE : Int;
      zero : Byte;
      status_sfc21 : Int;
      Error : Bool;
      status : Word;
   END_VAR
   VAR_TEMP   // added for the SCL form of the ladder/FBD networks
      _w1 : Bool;
   END_VAR
BEGIN

REGION Network 1: CALL FC2
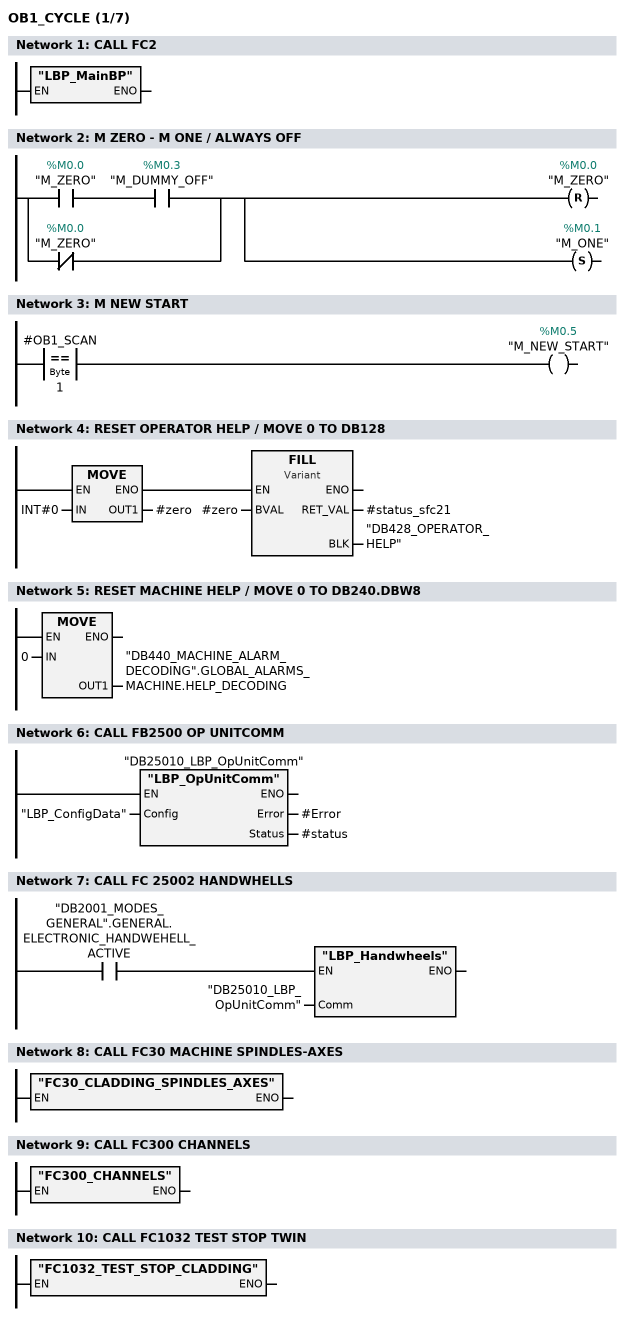
   RUNG wire#powerrail
      "LBP_MainBP"()
   END_RUNG
   // the same network as SCL:
   "LBP_MainBP"();
END_REGION

REGION Network 2: M ZERO - M ONE / ALWAYS OFF
   RUNG wire#powerrail
      Contact( "M_ZERO" )
      Contact( "M_DUMMY_OFF" )
      wire#w1
      R_Coil( "M_ZERO" )
   END_RUNG
   RUNG wire#powerrail
      I_Contact( "M_ZERO" )
   END_RUNG wire#w1
   RUNG wire#w1
      S_Coil( "M_ONE" )
   END_RUNG
   // the same network as SCL:
   #_w1 := ("M_ZERO" AND "M_DUMMY_OFF") OR NOT "M_ZERO";
   IF #_w1 THEN
       "M_ZERO" := FALSE;
       "M_ONE" := TRUE;
   END_IF;
END_REGION

REGION Network 3: M NEW START
   RUNG wire#powerrail
      { S7_Templates := "SrcType := Byte" } EQ_Contact(in1 := #OB1_SCAN, in2 := 1)
      Coil( "M_NEW_START" )
   END_RUNG
   // the same network as SCL:
   "M_NEW_START" := #OB1_SCAN = 1;
END_REGION

REGION Network 4: RESET OPERATOR HELP / MOVE 0 TO DB128
   RUNG wire#powerrail
      { S7_GenerateENO := "TRUE" } Move(in := INT#0, out1 => #zero)
      { S7_Templates := "ptr_type := Variant" } FILL(BVAL := #zero, RET_VAL => #status_sfc21, BLK => "DB428_OPERATOR_HELP")
   END_RUNG
   // the same network as SCL:
   // ENO of a box is taken as its EN; it also drops when the box reports an error
   #zero := INT#0;
   #status_sfc21 := FILL(BVAL := #zero, BLK => "DB428_OPERATOR_HELP");
END_REGION

REGION Network 5: RESET MACHINE HELP / MOVE 0 TO DB240.DBW8
   RUNG wire#powerrail
      { S7_GenerateENO := "TRUE" } Move(in := 0, out1 => "DB440_MACHINE_ALARM_DECODING".GLOBAL_ALARMS_MACHINE.HELP_DECODING)
   END_RUNG
   // the same network as SCL:
   "DB440_MACHINE_ALARM_DECODING".GLOBAL_ALARMS_MACHINE.HELP_DECODING := 0;
END_REGION

REGION Network 6: CALL FB2500 OP UNITCOMM
   RUNG wire#powerrail
      "DB25010_LBP_OpUnitComm"(Config := "LBP_ConfigData", Error => #Error, Status => #status)
   END_RUNG
   // the same network as SCL:
   "DB25010_LBP_OpUnitComm"(Config := "LBP_ConfigData", Error => #Error, Status => #status);   // "LBP_OpUnitComm"
END_REGION

REGION Network 7: CALL FC 25002 HANDWHELLS
   RUNG wire#powerrail
      Contact( "DB2001_MODES_GENERAL".GENERAL.ELECTRONIC_HANDWEHELL_ACTIVE )
      "LBP_Handwheels"(Comm := "DB25010_LBP_OpUnitComm")
   END_RUNG
   // the same network as SCL:
   IF "DB2001_MODES_GENERAL".GENERAL.ELECTRONIC_HANDWEHELL_ACTIVE THEN
       "LBP_Handwheels"(Comm := "DB25010_LBP_OpUnitComm");
   END_IF;
END_REGION

REGION Network 8: CALL FC30 MACHINE SPINDLES-AXES
   RUNG wire#powerrail
      "FC30_CLADDING_SPINDLES_AXES"()
   END_RUNG
   // the same network as SCL:
   "FC30_CLADDING_SPINDLES_AXES"();
END_REGION

REGION Network 9: CALL FC300 CHANNELS
   RUNG wire#powerrail
      "FC300_CHANNELS"()
   END_RUNG
   // the same network as SCL:
   "FC300_CHANNELS"();
END_REGION

REGION Network 10: CALL FC1032 TEST STOP TWIN
   RUNG wire#powerrail
      "FC1032_TEST_STOP_CLADDING"()
   END_RUNG
   // the same network as SCL:
   "FC1032_TEST_STOP_CLADDING"();
END_REGION

REGION Network 11: CALL FC1090 IDEVICE SI
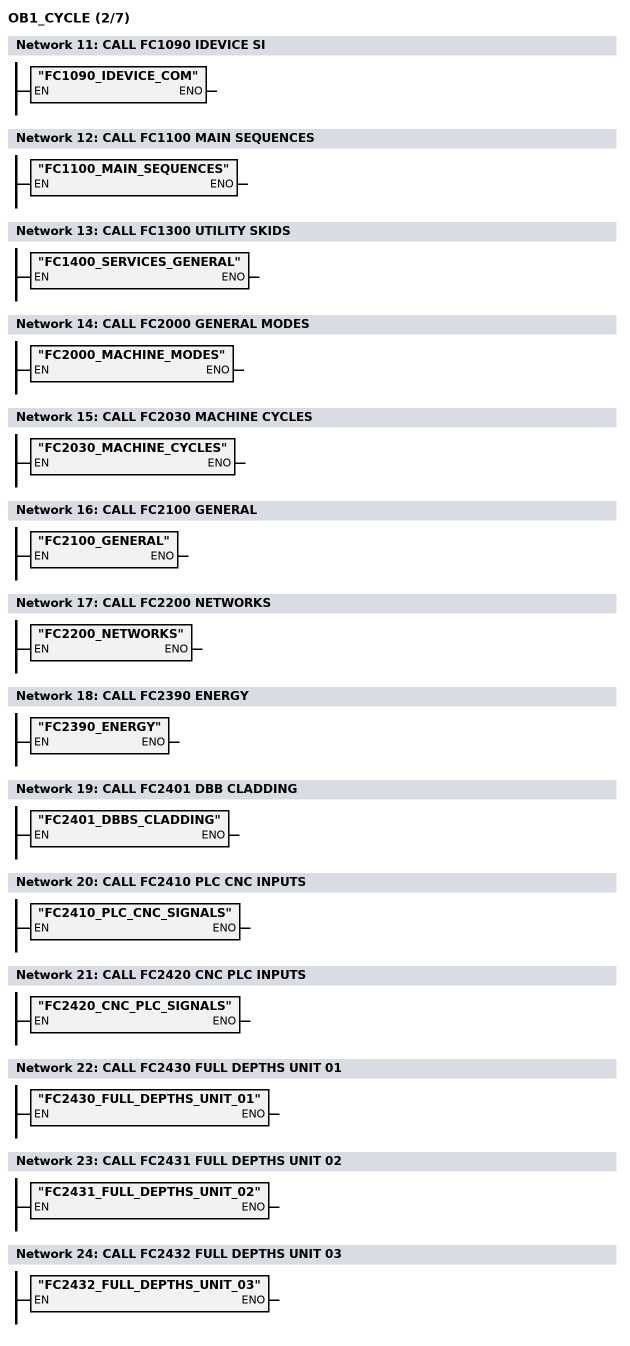
   RUNG wire#powerrail
      "FC1090_IDEVICE_COM"()
   END_RUNG
   // the same network as SCL:
   "FC1090_IDEVICE_COM"();
END_REGION

REGION Network 12: CALL FC1100 MAIN SEQUENCES
   RUNG wire#powerrail
      "FC1100_MAIN_SEQUENCES"()
   END_RUNG
   // the same network as SCL:
   "FC1100_MAIN_SEQUENCES"();
END_REGION

REGION Network 13: CALL FC1300 UTILITY SKIDS
   RUNG wire#powerrail
      "FC1400_SERVICES_GENERAL"()
   END_RUNG
   // the same network as SCL:
   "FC1400_SERVICES_GENERAL"();
END_REGION

REGION Network 14: CALL FC2000 GENERAL MODES
   RUNG wire#powerrail
      "FC2000_MACHINE_MODES"()
   END_RUNG
   // the same network as SCL:
   "FC2000_MACHINE_MODES"();
END_REGION

REGION Network 15: CALL FC2030 MACHINE CYCLES
   RUNG wire#powerrail
      "FC2030_MACHINE_CYCLES"()
   END_RUNG
   // the same network as SCL:
   "FC2030_MACHINE_CYCLES"();
END_REGION

REGION Network 16: CALL FC2100 GENERAL
   RUNG wire#powerrail
      "FC2100_GENERAL"()
   END_RUNG
   // the same network as SCL:
   "FC2100_GENERAL"();
END_REGION

REGION Network 17: CALL FC2200 NETWORKS
   RUNG wire#powerrail
      "FC2200_NETWORKS"()
   END_RUNG
   // the same network as SCL:
   "FC2200_NETWORKS"();
END_REGION

REGION Network 18: CALL FC2390 ENERGY
   RUNG wire#powerrail
      "FC2390_ENERGY"()
   END_RUNG
   // the same network as SCL:
   "FC2390_ENERGY"();
END_REGION

REGION Network 19: CALL FC2401 DBB CLADDING
   RUNG wire#powerrail
      "FC2401_DBBS_CLADDING"()
   END_RUNG
   // the same network as SCL:
   "FC2401_DBBS_CLADDING"();
END_REGION

REGION Network 20: CALL FC2410 PLC CNC INPUTS
   RUNG wire#powerrail
      "FC2410_PLC_CNC_SIGNALS"()
   END_RUNG
   // the same network as SCL:
   "FC2410_PLC_CNC_SIGNALS"();
END_REGION

REGION Network 21: CALL FC2420 CNC PLC INPUTS
   RUNG wire#powerrail
      "FC2420_CNC_PLC_SIGNALS"()
   END_RUNG
   // the same network as SCL:
   "FC2420_CNC_PLC_SIGNALS"();
END_REGION

REGION Network 22: CALL FC2430 FULL DEPTHS UNIT 01
   RUNG wire#powerrail
      "FC2430_FULL_DEPTHS_UNIT_01"()
   END_RUNG
   // the same network as SCL:
   "FC2430_FULL_DEPTHS_UNIT_01"();
END_REGION

REGION Network 23: CALL FC2431 FULL DEPTHS UNIT 02
   RUNG wire#powerrail
      "FC2431_FULL_DEPTHS_UNIT_02"()
   END_RUNG
   // the same network as SCL:
   "FC2431_FULL_DEPTHS_UNIT_02"();
END_REGION

REGION Network 24: CALL FC2432 FULL DEPTHS UNIT 03
   RUNG wire#powerrail
      "FC2432_FULL_DEPTHS_UNIT_03"()
   END_RUNG
   // the same network as SCL:
   "FC2432_FULL_DEPTHS_UNIT_03"();
END_REGION

REGION Network 25: CALL FC2440 GLOBAL DATA CLADDING
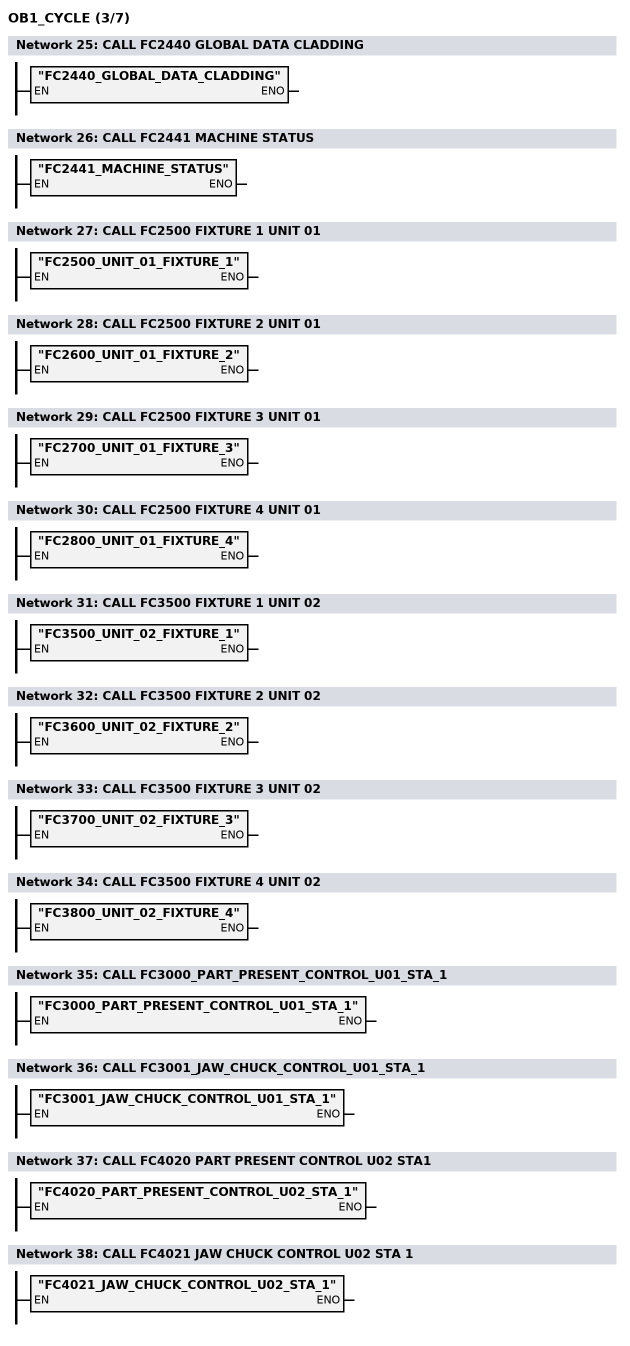
   RUNG wire#powerrail
      "FC2440_GLOBAL_DATA_CLADDING"()
   END_RUNG
   // the same network as SCL:
   "FC2440_GLOBAL_DATA_CLADDING"();
END_REGION

REGION Network 26: CALL FC2441 MACHINE STATUS
   RUNG wire#powerrail
      "FC2441_MACHINE_STATUS"()
   END_RUNG
   // the same network as SCL:
   "FC2441_MACHINE_STATUS"();
END_REGION

REGION Network 27: CALL FC2500 FIXTURE 1 UNIT 01
   RUNG wire#powerrail
      "FC2500_UNIT_01_FIXTURE_1"()
   END_RUNG
   // the same network as SCL:
   "FC2500_UNIT_01_FIXTURE_1"();
END_REGION

REGION Network 28: CALL FC2500 FIXTURE 2 UNIT 01
   RUNG wire#powerrail
      "FC2600_UNIT_01_FIXTURE_2"()
   END_RUNG
   // the same network as SCL:
   "FC2600_UNIT_01_FIXTURE_2"();
END_REGION

REGION Network 29: CALL FC2500 FIXTURE 3 UNIT 01
   RUNG wire#powerrail
      "FC2700_UNIT_01_FIXTURE_3"()
   END_RUNG
   // the same network as SCL:
   "FC2700_UNIT_01_FIXTURE_3"();
END_REGION

REGION Network 30: CALL FC2500 FIXTURE 4 UNIT 01
   RUNG wire#powerrail
      "FC2800_UNIT_01_FIXTURE_4"()
   END_RUNG
   // the same network as SCL:
   "FC2800_UNIT_01_FIXTURE_4"();
END_REGION

REGION Network 31: CALL FC3500 FIXTURE 1 UNIT 02
   RUNG wire#powerrail
      "FC3500_UNIT_02_FIXTURE_1"()
   END_RUNG
   // the same network as SCL:
   "FC3500_UNIT_02_FIXTURE_1"();
END_REGION

REGION Network 32: CALL FC3500 FIXTURE 2 UNIT 02
   RUNG wire#powerrail
      "FC3600_UNIT_02_FIXTURE_2"()
   END_RUNG
   // the same network as SCL:
   "FC3600_UNIT_02_FIXTURE_2"();
END_REGION

REGION Network 33: CALL FC3500 FIXTURE 3 UNIT 02
   RUNG wire#powerrail
      "FC3700_UNIT_02_FIXTURE_3"()
   END_RUNG
   // the same network as SCL:
   "FC3700_UNIT_02_FIXTURE_3"();
END_REGION

REGION Network 34: CALL FC3500 FIXTURE 4 UNIT 02
   RUNG wire#powerrail
      "FC3800_UNIT_02_FIXTURE_4"()
   END_RUNG
   // the same network as SCL:
   "FC3800_UNIT_02_FIXTURE_4"();
END_REGION

REGION Network 35: CALL FC3000_PART_PRESENT_CONTROL_U01_STA_1
   RUNG wire#powerrail
      "FC3000_PART_PRESENT_CONTROL_U01_STA_1"()
   END_RUNG
   // the same network as SCL:
   "FC3000_PART_PRESENT_CONTROL_U01_STA_1"();
END_REGION

REGION Network 36: CALL FC3001_JAW_CHUCK_CONTROL_U01_STA_1
   RUNG wire#powerrail
      "FC3001_JAW_CHUCK_CONTROL_U01_STA_1"()
   END_RUNG
   // the same network as SCL:
   "FC3001_JAW_CHUCK_CONTROL_U01_STA_1"();
END_REGION

REGION Network 37: CALL FC4020 PART PRESENT CONTROL U02 STA1
   RUNG wire#powerrail
      "FC4020_PART_PRESENT_CONTROL_U02_STA_1"()
   END_RUNG
   // the same network as SCL:
   "FC4020_PART_PRESENT_CONTROL_U02_STA_1"();
END_REGION

REGION Network 38: CALL FC4021 JAW CHUCK CONTROL U02 STA 1
   RUNG wire#powerrail
      "FC4021_JAW_CHUCK_CONTROL_U02_STA_1"()
   END_RUNG
   // the same network as SCL:
   "FC4021_JAW_CHUCK_CONTROL_U02_STA_1"();
END_REGION

REGION Network 39: CALL FC4000 FIXTURE TABLE POSITIONS
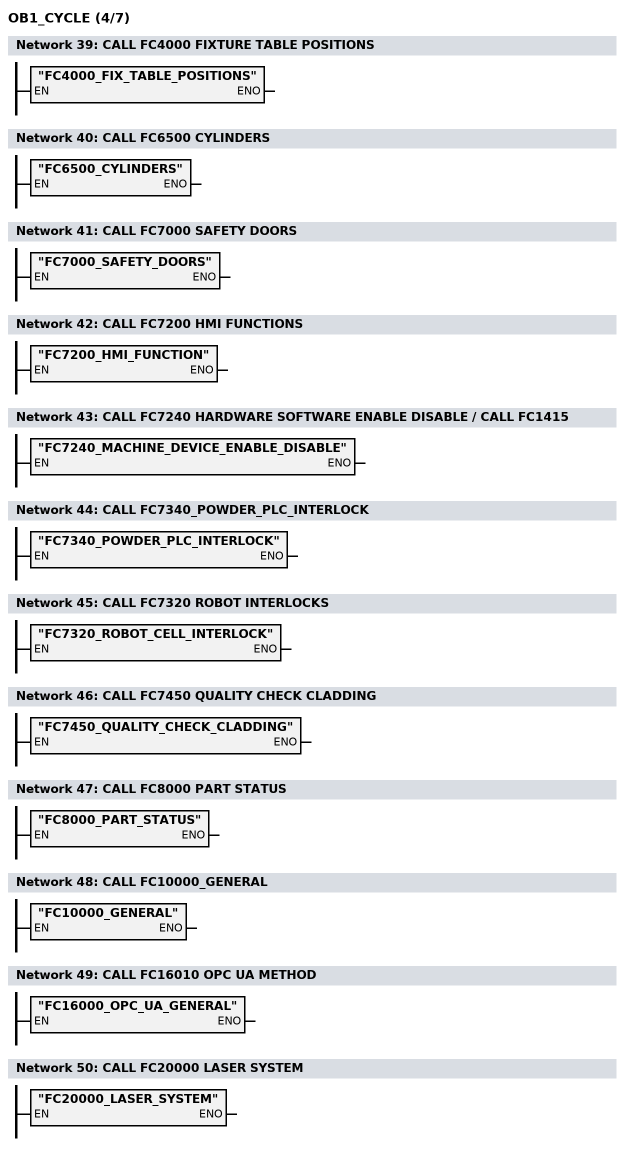
   RUNG wire#powerrail
      "FC4000_FIX_TABLE_POSITIONS"()
   END_RUNG
   // the same network as SCL:
   "FC4000_FIX_TABLE_POSITIONS"();
END_REGION

REGION Network 40: CALL FC6500 CYLINDERS
   RUNG wire#powerrail
      "FC6500_CYLINDERS"()
   END_RUNG
   // the same network as SCL:
   "FC6500_CYLINDERS"();
END_REGION

REGION Network 41: CALL FC7000 SAFETY DOORS
   RUNG wire#powerrail
      "FC7000_SAFETY_DOORS"()
   END_RUNG
   // the same network as SCL:
   "FC7000_SAFETY_DOORS"();
END_REGION

REGION Network 42: CALL FC7200 HMI FUNCTIONS
   RUNG wire#powerrail
      "FC7200_HMI_FUNCTION"()
   END_RUNG
   // the same network as SCL:
   "FC7200_HMI_FUNCTION"();
END_REGION

REGION Network 43: CALL FC7240 HARDWARE SOFTWARE ENABLE DISABLE / CALL FC1415
   RUNG wire#powerrail
      "FC7240_MACHINE_DEVICE_ENABLE_DISABLE"()
   END_RUNG
   // the same network as SCL:
   "FC7240_MACHINE_DEVICE_ENABLE_DISABLE"();
END_REGION

REGION Network 44: CALL FC7340_POWDER_PLC_INTERLOCK
   RUNG wire#powerrail
      "FC7340_POWDER_PLC_INTERLOCK"()
   END_RUNG
   // the same network as SCL:
   "FC7340_POWDER_PLC_INTERLOCK"();
END_REGION

REGION Network 45: CALL FC7320 ROBOT INTERLOCKS
   RUNG wire#powerrail
      "FC7320_ROBOT_CELL_INTERLOCK"()
   END_RUNG
   // the same network as SCL:
   "FC7320_ROBOT_CELL_INTERLOCK"();
END_REGION

REGION Network 46: CALL FC7450 QUALITY CHECK CLADDING
   RUNG wire#powerrail
      "FC7450_QUALITY_CHECK_CLADDING"()
   END_RUNG
   // the same network as SCL:
   "FC7450_QUALITY_CHECK_CLADDING"();
END_REGION

REGION Network 47: CALL FC8000 PART STATUS
   RUNG wire#powerrail
      "FC8000_PART_STATUS"()
   END_RUNG
   // the same network as SCL:
   "FC8000_PART_STATUS"();
END_REGION

REGION Network 48: CALL FC10000_GENERAL
   RUNG wire#powerrail
      "FC10000_GENERAL"()
   END_RUNG
   // the same network as SCL:
   "FC10000_GENERAL"();
END_REGION

REGION Network 49: CALL FC16010 OPC UA METHOD
   RUNG wire#powerrail
      "FC16000_OPC_UA_GENERAL"()
   END_RUNG
   // the same network as SCL:
   "FC16000_OPC_UA_GENERAL"();
END_REGION

REGION Network 50: CALL FC20000 LASER SYSTEM
   RUNG wire#powerrail
      "FC20000_LASER_SYSTEM"()
   END_RUNG
   // the same network as SCL:
   "FC20000_LASER_SYSTEM"();
END_REGION

REGION Network 51: SCREEN DARKENING
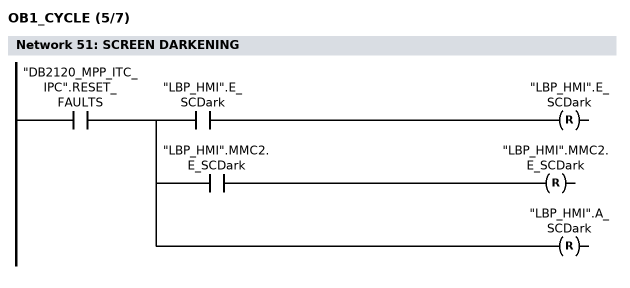
   RUNG wire#powerrail
      Contact( "DB2120_MPP_ITC_IPC".RESET_FAULTS )
      wire#w1
      Contact( "LBP_HMI".E_SCDark )
      R_Coil( "LBP_HMI".E_SCDark )
   END_RUNG
   RUNG wire#w1
      Contact( "LBP_HMI".MMC2.E_SCDark )
      R_Coil( "LBP_HMI".MMC2.E_SCDark )
   END_RUNG
   RUNG wire#w1
      R_Coil( "LBP_HMI".A_SCDark )
   END_RUNG
   // the same network as SCL:
   IF "DB2120_MPP_ITC_IPC".RESET_FAULTS AND "LBP_HMI".E_SCDark THEN "LBP_HMI".E_SCDark := FALSE; END_IF;
   IF "DB2120_MPP_ITC_IPC".RESET_FAULTS AND "LBP_HMI".MMC2.E_SCDark THEN
       "LBP_HMI".MMC2.E_SCDark := FALSE;
   END_IF;
   IF "DB2120_MPP_ITC_IPC".RESET_FAULTS THEN "LBP_HMI".A_SCDark := FALSE; END_IF;
END_REGION

REGION Network 52: OPERATOR HELP
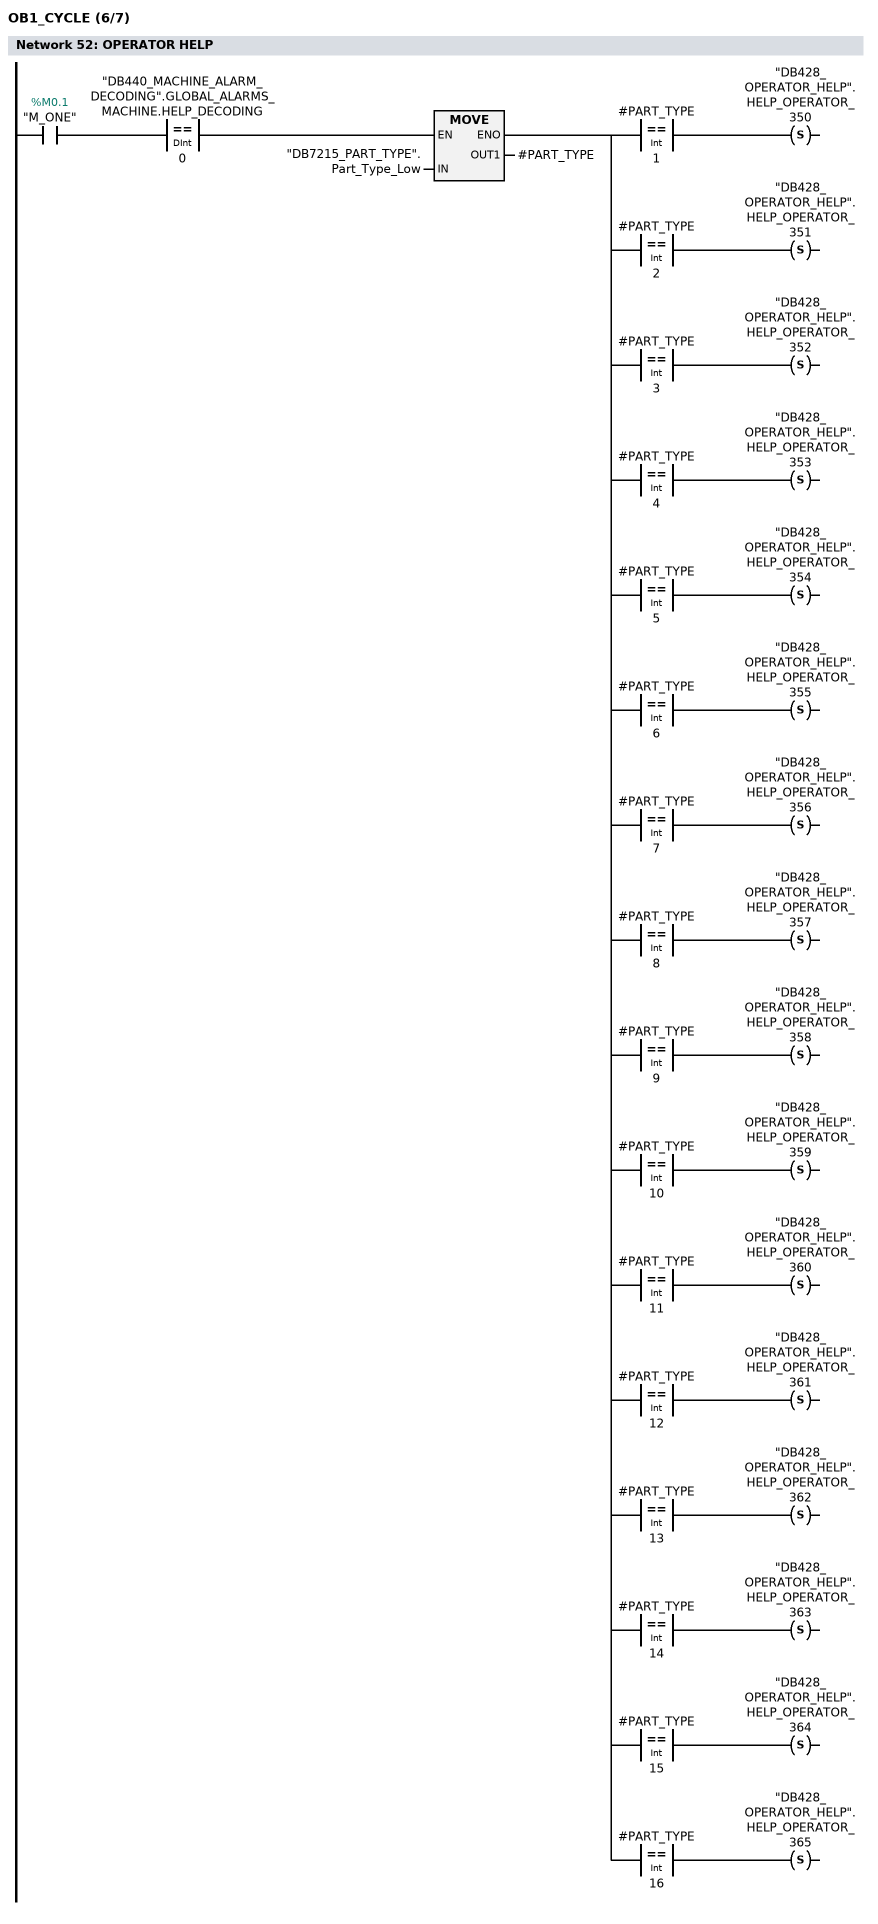
   RUNG wire#powerrail
      Contact( "M_ONE" )
      { S7_Templates := "SrcType := DInt" } EQ_Contact(in1 := "DB440_MACHINE_ALARM_DECODING".GLOBAL_ALARMS_MACHINE.HELP_DECODING, in2 := 0)
      { S7_GenerateENO := "TRUE" } Move(in := "DB7215_PART_TYPE".Part_Type_Low, out1 => #PART_TYPE)
      wire#w1
      { S7_Templates := "SrcType := Int" } EQ_Contact(in1 := #PART_TYPE, in2 := 1)
      S_Coil( "DB428_OPERATOR_HELP".HELP_OPERATOR_350 )
   END_RUNG
   RUNG wire#w1
      { S7_Templates := "SrcType := Int" } EQ_Contact(in1 := #PART_TYPE, in2 := 2)
      S_Coil( "DB428_OPERATOR_HELP".HELP_OPERATOR_351 )
   END_RUNG
   RUNG wire#w1
      { S7_Templates := "SrcType := Int" } EQ_Contact(in1 := #PART_TYPE, in2 := 3)
      S_Coil( "DB428_OPERATOR_HELP".HELP_OPERATOR_352 )
   END_RUNG
   RUNG wire#w1
      { S7_Templates := "SrcType := Int" } EQ_Contact(in1 := #PART_TYPE, in2 := 4)
      S_Coil( "DB428_OPERATOR_HELP".HELP_OPERATOR_353 )
   END_RUNG
   RUNG wire#w1
      { S7_Templates := "SrcType := Int" } EQ_Contact(in1 := #PART_TYPE, in2 := 5)
      S_Coil( "DB428_OPERATOR_HELP".HELP_OPERATOR_354 )
   END_RUNG
   RUNG wire#w1
      { S7_Templates := "SrcType := Int" } EQ_Contact(in1 := #PART_TYPE, in2 := 6)
      S_Coil( "DB428_OPERATOR_HELP".HELP_OPERATOR_355 )
   END_RUNG
   RUNG wire#w1
      { S7_Templates := "SrcType := Int" } EQ_Contact(in1 := #PART_TYPE, in2 := 7)
      S_Coil( "DB428_OPERATOR_HELP".HELP_OPERATOR_356 )
   END_RUNG
   RUNG wire#w1
      { S7_Templates := "SrcType := Int" } EQ_Contact(in1 := #PART_TYPE, in2 := 8)
      S_Coil( "DB428_OPERATOR_HELP".HELP_OPERATOR_357 )
   END_RUNG
   RUNG wire#w1
      { S7_Templates := "SrcType := Int" } EQ_Contact(in1 := #PART_TYPE, in2 := 9)
      S_Coil( "DB428_OPERATOR_HELP".HELP_OPERATOR_358 )
   END_RUNG
   RUNG wire#w1
      { S7_Templates := "SrcType := Int" } EQ_Contact(in1 := #PART_TYPE, in2 := 10)
      S_Coil( "DB428_OPERATOR_HELP".HELP_OPERATOR_359 )
   END_RUNG
   RUNG wire#w1
      { S7_Templates := "SrcType := Int" } EQ_Contact(in1 := #PART_TYPE, in2 := 11)
      S_Coil( "DB428_OPERATOR_HELP".HELP_OPERATOR_360 )
   END_RUNG
   RUNG wire#w1
      { S7_Templates := "SrcType := Int" } EQ_Contact(in1 := #PART_TYPE, in2 := 12)
      S_Coil( "DB428_OPERATOR_HELP".HELP_OPERATOR_361 )
   END_RUNG
   RUNG wire#w1
      { S7_Templates := "SrcType := Int" } EQ_Contact(in1 := #PART_TYPE, in2 := 13)
      S_Coil( "DB428_OPERATOR_HELP".HELP_OPERATOR_362 )
   END_RUNG
   RUNG wire#w1
      { S7_Templates := "SrcType := Int" } EQ_Contact(in1 := #PART_TYPE, in2 := 14)
      S_Coil( "DB428_OPERATOR_HELP".HELP_OPERATOR_363 )
   END_RUNG
   RUNG wire#w1
      { S7_Templates := "SrcType := Int" } EQ_Contact(in1 := #PART_TYPE, in2 := 15)
      S_Coil( "DB428_OPERATOR_HELP".HELP_OPERATOR_364 )
   END_RUNG
   RUNG wire#w1
      { S7_Templates := "SrcType := Int" } EQ_Contact(in1 := #PART_TYPE, in2 := 16)
      S_Coil( "DB428_OPERATOR_HELP".HELP_OPERATOR_365 )
   END_RUNG
   // the same network as SCL:
   // ENO of a box is taken as its EN; it also drops when the box reports an error
   #_w1 := "M_ONE" AND ("DB440_MACHINE_ALARM_DECODING".GLOBAL_ALARMS_MACHINE.HELP_DECODING = 0);
   IF #_w1 THEN #PART_TYPE := "DB7215_PART_TYPE".Part_Type_Low; END_IF;
   IF #_w1 AND (#PART_TYPE = 1) THEN "DB428_OPERATOR_HELP".HELP_OPERATOR_350 := TRUE; END_IF;
   IF #_w1 AND (#PART_TYPE = 2) THEN "DB428_OPERATOR_HELP".HELP_OPERATOR_351 := TRUE; END_IF;
   IF #_w1 AND (#PART_TYPE = 3) THEN "DB428_OPERATOR_HELP".HELP_OPERATOR_352 := TRUE; END_IF;
   IF #_w1 AND (#PART_TYPE = 4) THEN "DB428_OPERATOR_HELP".HELP_OPERATOR_353 := TRUE; END_IF;
   IF #_w1 AND (#PART_TYPE = 5) THEN "DB428_OPERATOR_HELP".HELP_OPERATOR_354 := TRUE; END_IF;
   IF #_w1 AND (#PART_TYPE = 6) THEN "DB428_OPERATOR_HELP".HELP_OPERATOR_355 := TRUE; END_IF;
   IF #_w1 AND (#PART_TYPE = 7) THEN "DB428_OPERATOR_HELP".HELP_OPERATOR_356 := TRUE; END_IF;
   IF #_w1 AND (#PART_TYPE = 8) THEN "DB428_OPERATOR_HELP".HELP_OPERATOR_357 := TRUE; END_IF;
   IF #_w1 AND (#PART_TYPE = 9) THEN "DB428_OPERATOR_HELP".HELP_OPERATOR_358 := TRUE; END_IF;
   IF #_w1 AND (#PART_TYPE = 10) THEN "DB428_OPERATOR_HELP".HELP_OPERATOR_359 := TRUE; END_IF;
   IF #_w1 AND (#PART_TYPE = 11) THEN "DB428_OPERATOR_HELP".HELP_OPERATOR_360 := TRUE; END_IF;
   IF #_w1 AND (#PART_TYPE = 12) THEN "DB428_OPERATOR_HELP".HELP_OPERATOR_361 := TRUE; END_IF;
   IF #_w1 AND (#PART_TYPE = 13) THEN "DB428_OPERATOR_HELP".HELP_OPERATOR_362 := TRUE; END_IF;
   IF #_w1 AND (#PART_TYPE = 14) THEN "DB428_OPERATOR_HELP".HELP_OPERATOR_363 := TRUE; END_IF;
   IF #_w1 AND (#PART_TYPE = 15) THEN "DB428_OPERATOR_HELP".HELP_OPERATOR_364 := TRUE; END_IF;
   IF #_w1 AND (#PART_TYPE = 16) THEN "DB428_OPERATOR_HELP".HELP_OPERATOR_365 := TRUE; END_IF;
END_REGION

REGION Network 53: CALL FC428 OPERATOR HELP
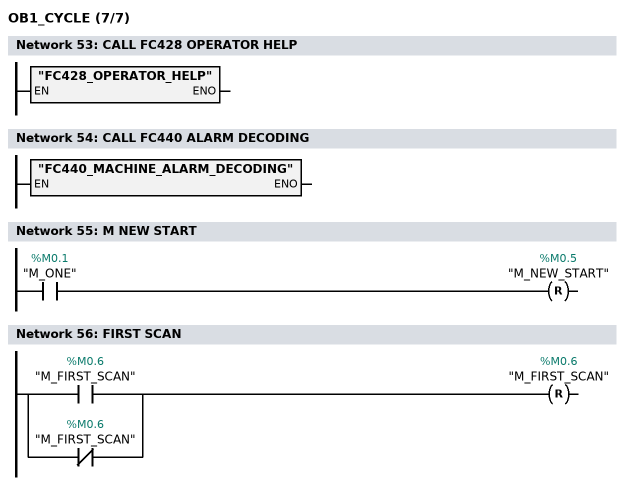
   RUNG wire#powerrail
      "FC428_OPERATOR_HELP"()
   END_RUNG
   // the same network as SCL:
   "FC428_OPERATOR_HELP"();
END_REGION

REGION Network 54: CALL FC440 ALARM DECODING
   RUNG wire#powerrail
      "FC440_MACHINE_ALARM_DECODING"()
   END_RUNG
   // the same network as SCL:
   "FC440_MACHINE_ALARM_DECODING"();
END_REGION

REGION Network 55: M NEW START
   RUNG wire#powerrail
      Contact( "M_ONE" )
      R_Coil( "M_NEW_START" )
   END_RUNG
   // the same network as SCL:
   IF "M_ONE" THEN "M_NEW_START" := FALSE; END_IF;
END_REGION

REGION Network 56: FIRST SCAN
   RUNG wire#powerrail
      Contact( "M_FIRST_SCAN" )
      wire#w1
      R_Coil( "M_FIRST_SCAN" )
   END_RUNG
   RUNG wire#powerrail
      I_Contact( "M_FIRST_SCAN" )
   END_RUNG wire#w1
   // the same network as SCL:
   IF "M_FIRST_SCAN" OR NOT "M_FIRST_SCAN" THEN "M_FIRST_SCAN" := FALSE; END_IF;
END_REGION
END_ORGANIZATION_BLOCK

FUNCTION "FC300_CHANNELS" : Void   // FC300, LAD
{ S7_Optimized_Access := 'FALSE' }
AUTHOR : ETXETAR
VERSION : 1.0
// stored: AutoNumber false, IsIECCheckEnabled false, SetENOAutomatically false, UDAEnableTagReadback false
BEGIN

REGION Network 1: CALL FC321 CHANNEL 1 / CALL FC121
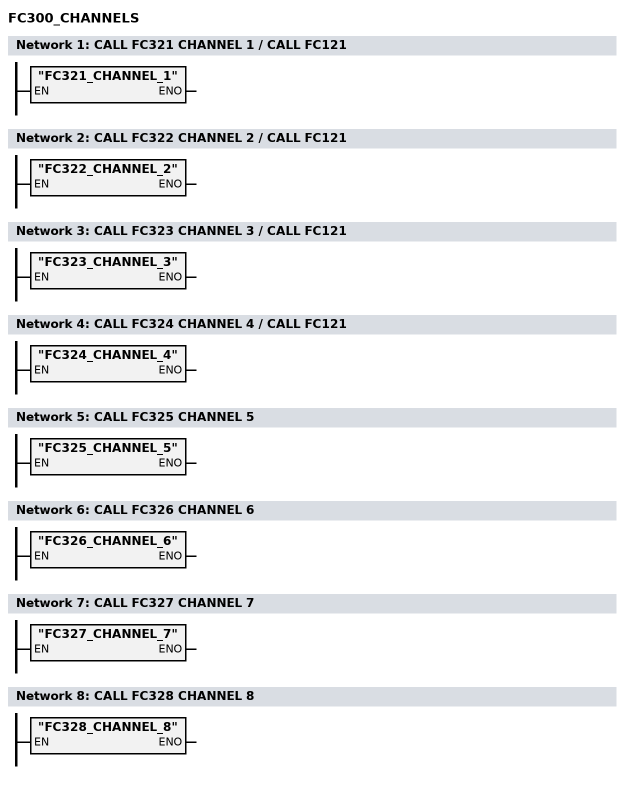
   RUNG wire#powerrail
      "FC321_CHANNEL_1"()
   END_RUNG
   // the same network as SCL:
   "FC321_CHANNEL_1"();
END_REGION

REGION Network 2: CALL FC322 CHANNEL 2 / CALL FC121
   RUNG wire#powerrail
      "FC322_CHANNEL_2"()
   END_RUNG
   // the same network as SCL:
   "FC322_CHANNEL_2"();
END_REGION

REGION Network 3: CALL FC323 CHANNEL 3 / CALL FC121
   RUNG wire#powerrail
      "FC323_CHANNEL_3"()
   END_RUNG
   // the same network as SCL:
   "FC323_CHANNEL_3"();
END_REGION

REGION Network 4: CALL FC324 CHANNEL 4 / CALL FC121
   RUNG wire#powerrail
      "FC324_CHANNEL_4"()
   END_RUNG
   // the same network as SCL:
   "FC324_CHANNEL_4"();
END_REGION

REGION Network 5: CALL FC325 CHANNEL 5
   RUNG wire#powerrail
      "FC325_CHANNEL_5"()
   END_RUNG
   // the same network as SCL:
   "FC325_CHANNEL_5"();
END_REGION

REGION Network 6: CALL FC326 CHANNEL 6
   RUNG wire#powerrail
      "FC326_CHANNEL_6"()
   END_RUNG
   // the same network as SCL:
   "FC326_CHANNEL_6"();
END_REGION

REGION Network 7: CALL FC327 CHANNEL 7
   RUNG wire#powerrail
      "FC327_CHANNEL_7"()
   END_RUNG
   // the same network as SCL:
   "FC327_CHANNEL_7"();
END_REGION

REGION Network 8: CALL FC328 CHANNEL 8
   RUNG wire#powerrail
      "FC328_CHANNEL_8"()
   END_RUNG
   // the same network as SCL:
   "FC328_CHANNEL_8"();
END_REGION
END_FUNCTION

FUNCTION "FC1100_MAIN_SEQUENCES" : Void   // FC1100, LAD
{ S7_Optimized_Access := 'FALSE' }
AUTHOR : ETXETAR
VERSION : 1.0
// stored: AutoNumber false, IsIECCheckEnabled false, SetENOAutomatically false, UDAEnableTagReadback false
   VAR_TEMP
      STEP_NUMBER : Int;
   END_VAR
BEGIN

REGION Network 1: CALL FC1103 MACHINING TWIN TWIN+
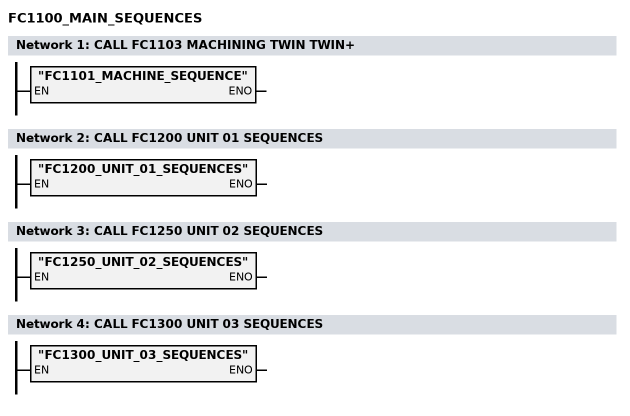
   RUNG wire#powerrail
      "FC1101_MACHINE_SEQUENCE"()
   END_RUNG
   // the same network as SCL:
   "FC1101_MACHINE_SEQUENCE"();
END_REGION

REGION Network 2: CALL FC1200 UNIT 01 SEQUENCES
   RUNG wire#powerrail
      "FC1200_UNIT_01_SEQUENCES"()
   END_RUNG
   // the same network as SCL:
   "FC1200_UNIT_01_SEQUENCES"();
END_REGION

REGION Network 3: CALL FC1250 UNIT 02 SEQUENCES
   RUNG wire#powerrail
      "FC1250_UNIT_02_SEQUENCES"()
   END_RUNG
   // the same network as SCL:
   "FC1250_UNIT_02_SEQUENCES"();
END_REGION

REGION Network 4: CALL FC1300 UNIT 03 SEQUENCES
   RUNG wire#powerrail
      "FC1300_UNIT_03_SEQUENCES"()
   END_RUNG
   // the same network as SCL:
   "FC1300_UNIT_03_SEQUENCES"();
END_REGION
END_FUNCTION

FUNCTION "FC1400_SERVICES_GENERAL" : Void   // FC1400, LAD
{ S7_Optimized_Access := 'FALSE' }
AUTHOR : ETXETAR
VERSION : 1.0
// stored: AutoNumber false, IsIECCheckEnabled false, SetENOAutomatically false, UDAEnableTagReadback false
BEGIN

REGION Network 1: CALL FC1401_UTILITY_SKIDS
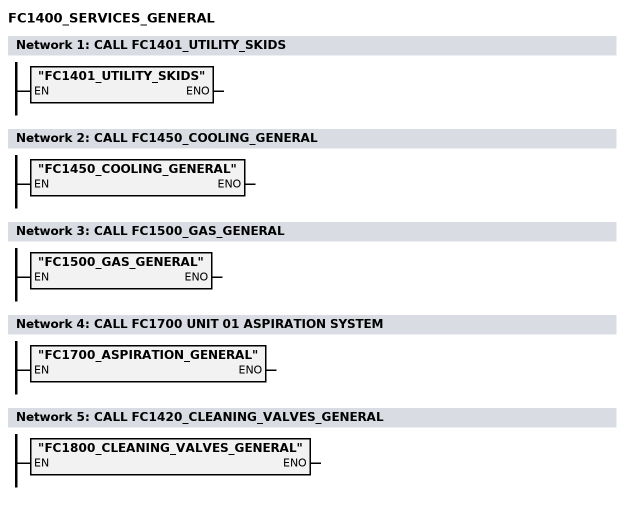
   RUNG wire#powerrail
      "FC1401_UTILITY_SKIDS"()
   END_RUNG
   // the same network as SCL:
   "FC1401_UTILITY_SKIDS"();
END_REGION

REGION Network 2: CALL FC1450_COOLING_GENERAL
   RUNG wire#powerrail
      "FC1450_COOLING_GENERAL"()
   END_RUNG
   // the same network as SCL:
   "FC1450_COOLING_GENERAL"();
END_REGION

REGION Network 3: CALL FC1500_GAS_GENERAL
   RUNG wire#powerrail
      "FC1500_GAS_GENERAL"()
   END_RUNG
   // the same network as SCL:
   "FC1500_GAS_GENERAL"();
END_REGION

REGION Network 4: CALL FC1700 UNIT 01 ASPIRATION SYSTEM
   RUNG wire#powerrail
      "FC1700_ASPIRATION_GENERAL"()
   END_RUNG
   // the same network as SCL:
   "FC1700_ASPIRATION_GENERAL"();
END_REGION

REGION Network 5: CALL FC1420_CLEANING_VALVES_GENERAL
   RUNG wire#powerrail
      "FC1800_CLEANING_VALVES_GENERAL"()
   END_RUNG
   // the same network as SCL:
   "FC1800_CLEANING_VALVES_GENERAL"();
END_REGION
END_FUNCTION

FUNCTION "FC1401_UTILITY_SKIDS" : Void   // FC1401, LAD
{ S7_Optimized_Access := 'TRUE' }
VERSION : 0.1
// stored: AutoNumber false, IsIECCheckEnabled false, SetENOAutomatically false, UDAEnableTagReadback false
   VAR CONSTANT
      FC_NUMBER : DInt := 1401;
   END_VAR
   VAR_TEMP   // added for the SCL form of the ladder/FBD networks
      _w1 : Bool;
      _w2 : Bool;
   END_VAR
BEGIN

REGION Network 1: <<<<<<<<<<<<<<<<<<<< PNEUMATIC SYSTEM >>>>>>>>>>>>>>>>>>>>
END_REGION

REGION Network 2: CALL FB1401 PNEUMATIC SYSTEM
   // 2#0000_0001 OPTIONS 0 BIT 0 PRESSURE PRESENT OPTION
   // 2#0000_0010 OPTIONS 0 BIT 1 CONNECTION SENSOR 1 OPTION
   // 2#0000_0100 OPTIONS 0 BIT 2 CONNECTION SENSOR 2 OPTION
   // 2#0000_1000 OPTIONS 0 BIT 3 DRIVE UNBLOCKED OPTION
   // 2#0001_0000 OPTIONS 0 BIT 4 PRESSURIZED OPTION
   // 2#0010_0000 OPTIONS 0 BIT 5 UNIT 01 GRIPPER PRESSURIZED OPTION
   // 2#0100_0000 OPTIONS 0 BIT 6 UNIT 01 LABERINT PRESSURIZED OPTION
   // 2#1000_0000 OPTIONS 0 BIT 7 UNIT 01 UPPER TABLE PRESSURIZED OPTION
   // 
   // 2#0000_0001 OPTIONS 1 BIT 0 UNIT 01 LOWER TABLE PRESSURIZED OPTION
   // 2#0000_0010 OPTIONS 1 BIT 1 UNIT 01 AXIS X CART PRESSURIZED OPTION
   // 2#0000_0100 OPTIONS 1 BIT 2 UNIT 01 STATION 3 MEASURMENT UNIT PRESSURIZED OPTION
   // 2#0000_1000 OPTIONS 1 BIT 3 UNIT 01 STATION 4 MEASURMENT UNIT PRESSURIZED OPTION
   // 2#0001_0000 OPTIONS 1 BIT 4 UNIT 02 GRIPPER PRESSURIZEDPRESSURIZED OPTION
   // 2#0010_0000 OPTIONS 1 BIT 5 UNIT 02 LABERINT PRESSURIZED OPTION
   // 2#0100_0000 OPTIONS 1 BIT 6 UNIT 02 UPPER TABLE PRESSURIZED OPTION
   // 2#1000_0000 OPTIONS 1 BIT 7 UNIT 02 LOWER TABLE PRESSURIZED OPTION
   // 
   // 2#0000_0001 OPTIONS 2 BIT 0 UNIT 02 AXIS X CART PRESSURIZED OPTION
   // 2#0000_0010 OPTIONS 2 BIT 1 UNIT 02 STATION 3 MEASURMENT UNIT PRESSURIZED OPTION
   // 2#0000_0100 OPTIONS 2 BIT 2 UNIT 02 STATION 4 MEASURMENT UNIT PRESSURIZED OPTION
   // 2#0000_1000 OPTIONS 2 BIT 3 INPUT FLOW  OPTION
   // 2#0001_0000 OPTIONS 2 BIT 4 INPUT TEMPERATURE OPTION
   // 2#0010_0000 OPTIONS 2 BIT 5 SPARE OPTION
   // 2#0100_0000 OPTIONS 2 BIT 6 SPARE OPTION
   // 2#1000_0000 OPTIONS 2 BIT 7 SPARE OPTION
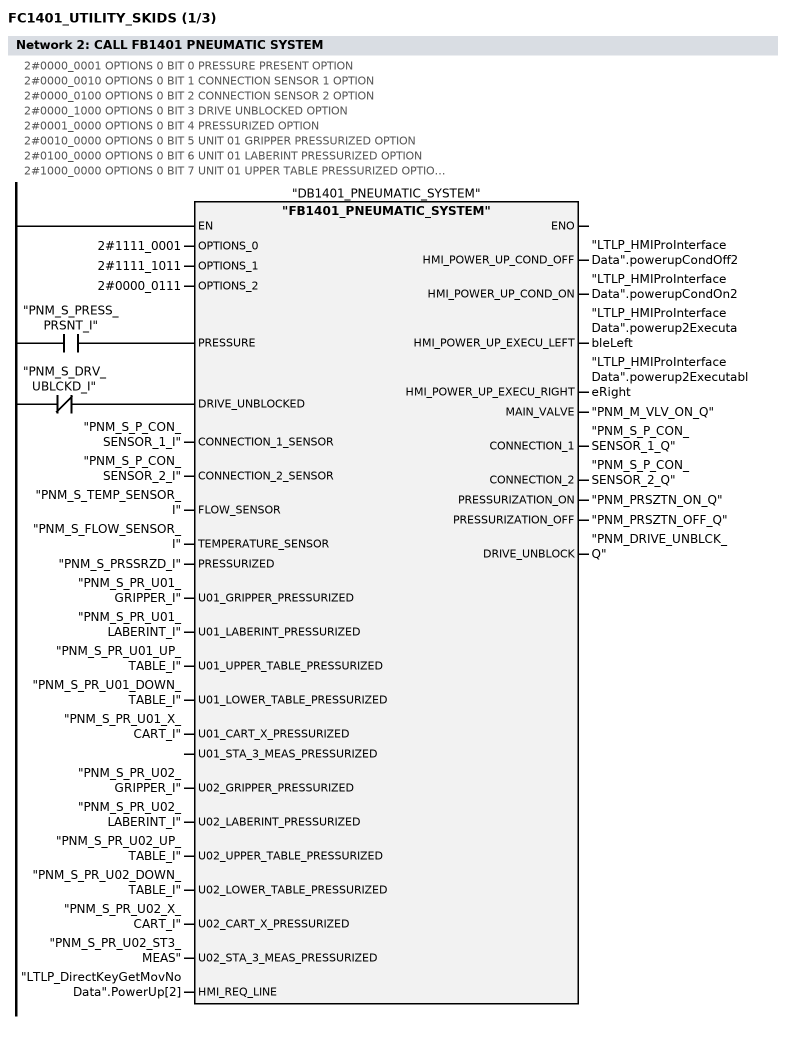
   RUNG wire#powerrail
      "DB1401_PNEUMATIC_SYSTEM"(PRESSURE := wire#w1, DRIVE_UNBLOCKED := wire#w2, OPTIONS_0 := 2#1111_0001, OPTIONS_1 := 2#1111_1011, OPTIONS_2 := 2#0000_0111, CONNECTION_1_SENSOR := "PNM_S_P_CON_SENSOR_1_I", CONNECTION_2_SENSOR := "PNM_S_P_CON_SENSOR_2_I", FLOW_SENSOR := "PNM_S_TEMP_SENSOR_I", TEMPERATURE_SENSOR := "PNM_S_FLOW_SENSOR_I", PRESSURIZED := "PNM_S_PRSSRZD_I", U01_GRIPPER_PRESSURIZED := "PNM_S_PR_U01_GRIPPER_I", U01_LABERINT_PRESSURIZED := "PNM_S_PR_U01_LABERINT_I", U01_UPPER_TABLE_PRESSURIZED := "PNM_S_PR_U01_UP_TABLE_I", U01_LOWER_TABLE_PRESSURIZED := "PNM_S_PR_U01_DOWN_TABLE_I", U01_CART_X_PRESSURIZED := "PNM_S_PR_U01_X_CART_I", U01_STA_3_MEAS_PRESSURIZED :=, U02_GRIPPER_PRESSURIZED := "PNM_S_PR_U02_GRIPPER_I", U02_LABERINT_PRESSURIZED := "PNM_S_PR_U02_LABERINT_I", U02_UPPER_TABLE_PRESSURIZED := "PNM_S_PR_U02_UP_TABLE_I", U02_LOWER_TABLE_PRESSURIZED := "PNM_S_PR_U02_DOWN_TABLE_I", U02_CART_X_PRESSURIZED := "PNM_S_PR_U02_X_CART_I", U02_STA_3_MEAS_PRESSURIZED := "PNM_S_PR_U02_ST3_MEAS", HMI_REQ_LINE := "LTLP_DirectKeyGetMovNoData".PowerUp[2], HMI_POWER_UP_COND_OFF => "LTLP_HMIProInterfaceData".powerupCondOff2, HMI_POWER_UP_COND_ON => "LTLP_HMIProInterfaceData".powerupCondOn2, HMI_POWER_UP_EXECU_LEFT => "LTLP_HMIProInterfaceData".powerup2ExecutableLeft, HMI_POWER_UP_EXECU_RIGHT => "LTLP_HMIProInterfaceData".powerup2ExecutableRight, MAIN_VALVE => "PNM_M_VLV_ON_Q", CONNECTION_1 => "PNM_S_P_CON_SENSOR_1_Q", CONNECTION_2 => "PNM_S_P_CON_SENSOR_2_Q", PRESSURIZATION_ON => "PNM_PRSZTN_ON_Q", PRESSURIZATION_OFF => "PNM_PRSZTN_OFF_Q", DRIVE_UNBLOCK => "PNM_DRIVE_UNBLCK_Q")
   END_RUNG
   RUNG wire#powerrail
      Contact( "PNM_S_PRESS_PRSNT_I" )
   END_RUNG wire#w1
   RUNG wire#powerrail
      I_Contact( "PNM_S_DRV_UBLCKD_I" )
   END_RUNG wire#w2
   // the same network as SCL:
   "DB1401_PNEUMATIC_SYSTEM"(OPTIONS_0 := 2#1111_0001,   // "FB1401_PNEUMATIC_SYSTEM"
                           OPTIONS_1 := 2#1111_1011,
                           OPTIONS_2 := 2#0000_0111,
                           PRESSURE := "PNM_S_PRESS_PRSNT_I",
                           DRIVE_UNBLOCKED := NOT "PNM_S_DRV_UBLCKD_I",
                           CONNECTION_1_SENSOR := "PNM_S_P_CON_SENSOR_1_I",
                           CONNECTION_2_SENSOR := "PNM_S_P_CON_SENSOR_2_I",
                           FLOW_SENSOR := "PNM_S_TEMP_SENSOR_I",
                           TEMPERATURE_SENSOR := "PNM_S_FLOW_SENSOR_I",
                           PRESSURIZED := "PNM_S_PRSSRZD_I",
                           U01_GRIPPER_PRESSURIZED := "PNM_S_PR_U01_GRIPPER_I",
                           U01_LABERINT_PRESSURIZED := "PNM_S_PR_U01_LABERINT_I",
                           U01_UPPER_TABLE_PRESSURIZED := "PNM_S_PR_U01_UP_TABLE_I",
                           U01_LOWER_TABLE_PRESSURIZED := "PNM_S_PR_U01_DOWN_TABLE_I",
                           U01_CART_X_PRESSURIZED := "PNM_S_PR_U01_X_CART_I",
                           U02_GRIPPER_PRESSURIZED := "PNM_S_PR_U02_GRIPPER_I",
                           U02_LABERINT_PRESSURIZED := "PNM_S_PR_U02_LABERINT_I",
                           U02_UPPER_TABLE_PRESSURIZED := "PNM_S_PR_U02_UP_TABLE_I",
                           U02_LOWER_TABLE_PRESSURIZED := "PNM_S_PR_U02_DOWN_TABLE_I",
                           U02_CART_X_PRESSURIZED := "PNM_S_PR_U02_X_CART_I",
                           U02_STA_3_MEAS_PRESSURIZED := "PNM_S_PR_U02_ST3_MEAS",
                           HMI_REQ_LINE := "LTLP_DirectKeyGetMovNoData".PowerUp[2],
                           HMI_POWER_UP_COND_OFF => "LTLP_HMIProInterfaceData".powerupCondOff2,
                           HMI_POWER_UP_COND_ON => "LTLP_HMIProInterfaceData".powerupCondOn2,
                           HMI_POWER_UP_EXECU_LEFT => "LTLP_HMIProInterfaceData".powerup2ExecutableLeft,
                           HMI_POWER_UP_EXECU_RIGHT => "LTLP_HMIProInterfaceData".powerup2ExecutableRight,
                           MAIN_VALVE => "PNM_M_VLV_ON_Q",
                           CONNECTION_1 => "PNM_S_P_CON_SENSOR_1_Q",
                           CONNECTION_2 => "PNM_S_P_CON_SENSOR_2_Q",
                           PRESSURIZATION_ON => "PNM_PRSZTN_ON_Q",
                           PRESSURIZATION_OFF => "PNM_PRSZTN_OFF_Q",
                           DRIVE_UNBLOCK => "PNM_DRIVE_UNBLCK_Q");
END_REGION

REGION Network 3: <<<<<<<<<<<<<<<<<<<< LUBRICATION SYSTEM >>>>>>>>>>>>>>>>>>>>
END_REGION

REGION Network 4: CALL FB1421 PROGRESSIVE LUBRICATION WITH GREASE
   // 2#0000_0001 OPTIONS 0 BIT 0 CIRCUIT BREAKER OPTION
   // 2#0000_0010 OPTIONS 0 BIT 1 LOW LEVEL ALARM OPTION
   // 2#0000_0100 OPTIONS 0 BIT 2 OVERPRESSURE ALARM OPTION
   // 2#0000_1000 OPTIONS 0 BIT 3 LUBRICATION BY TIME VALVE 1 AXIS X OPTION
   // 2#0001_0000 OPTIONS 0 BIT 4 LUBRICATION BY TIME VALVE 2 AXIS Z OPTION
   // 2#0010_0000 OPTIONS 0 BIT 5 LUBRICATION BY TIME VALVE 3 TURN UNIT OPTION
   // 2#0100_0000 OPTIONS 0 BIT 6 LUBRICATION BY TIME VALVE 4 OPTION
   // 2#1000_0000 OPTIONS 0 BIT 7 LUBRICATION DONE VALVE 1  AXIS X OPTION
   // 
   // 2#0000_0001 OPTIONS 1 BIT 0 LUBRICATION DONE VALVE 2 AXIS Z OPTION
   // 2#0000_0010 OPTIONS 1 BIT 1 LUBRICATION DONE VALVE 3 TURN UNIT OPTION
   // 2#0000_0100 OPTIONS 1 BIT 2 LUBRICATION DONE VALVE 4 OPTION
   // 2#0000_1000 OPTIONS 1 BIT 3 LUBRICATION DONE VALVE 5 OPTION
   // 2#0001_0000 OPTIONS 1 BIT 4 LUBRICATION DONE VALVE 6 OPTION
   // 2#0010_0000 OPTIONS 1 BIT 5 LUBRICATION DONE VALVE 7 OPTION
   // 2#0100_0000 OPTIONS 1 BIT 6 LUBRICATION DONE VALVE 8 OPTION
   // 2#1000_0000 OPTIONS 1 BIT 7 LUBRICATION DONE VALVE 9 OPTION
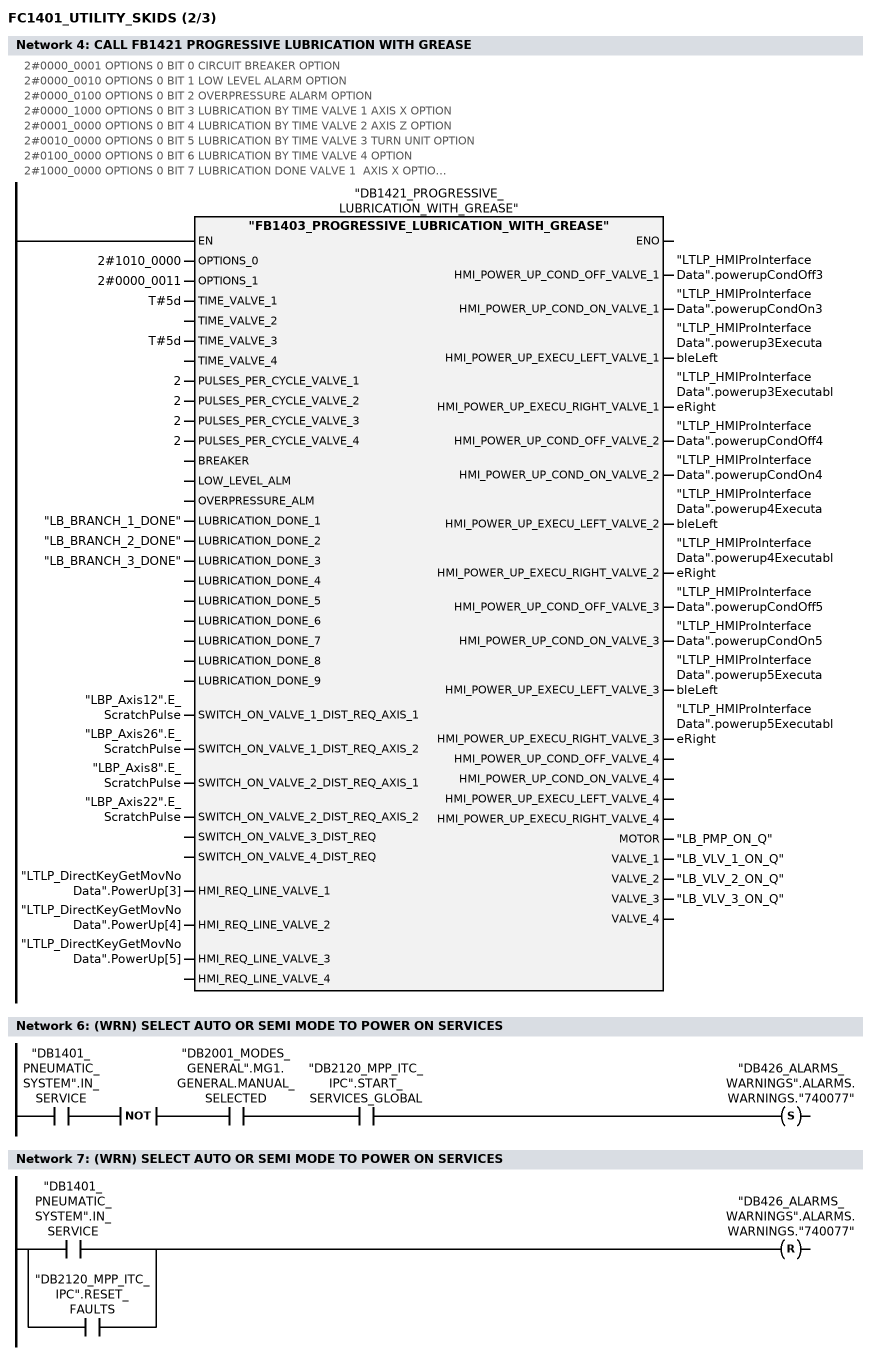
   RUNG wire#powerrail
      "DB1421_PROGRESSIVE_LUBRICATION_WITH_GREASE"(OPTIONS_0 := 2#1010_0000, OPTIONS_1 := 2#0000_0011, TIME_VALVE_1 := T#5d, TIME_VALVE_2 :=, TIME_VALVE_3 := T#5d, TIME_VALVE_4 :=, PULSES_PER_CYCLE_VALVE_1 := 2, PULSES_PER_CYCLE_VALVE_2 := 2, PULSES_PER_CYCLE_VALVE_3 := 2, PULSES_PER_CYCLE_VALVE_4 := 2, BREAKER :=, LOW_LEVEL_ALM :=, OVERPRESSURE_ALM :=, LUBRICATION_DONE_1 := "LB_BRANCH_1_DONE", LUBRICATION_DONE_2 := "LB_BRANCH_2_DONE", LUBRICATION_DONE_3 := "LB_BRANCH_3_DONE", LUBRICATION_DONE_4 :=, LUBRICATION_DONE_5 :=, LUBRICATION_DONE_6 :=, LUBRICATION_DONE_7 :=, LUBRICATION_DONE_8 :=, LUBRICATION_DONE_9 :=, SWITCH_ON_VALVE_1_DIST_REQ_AXIS_1 := "LBP_Axis12".E_ScratchPulse, SWITCH_ON_VALVE_1_DIST_REQ_AXIS_2 := "LBP_Axis26".E_ScratchPulse, SWITCH_ON_VALVE_2_DIST_REQ_AXIS_1 := "LBP_Axis8".E_ScratchPulse, SWITCH_ON_VALVE_2_DIST_REQ_AXIS_2 := "LBP_Axis22".E_ScratchPulse, SWITCH_ON_VALVE_3_DIST_REQ :=, SWITCH_ON_VALVE_4_DIST_REQ :=, HMI_REQ_LINE_VALVE_1 := "LTLP_DirectKeyGetMovNoData".PowerUp[3], HMI_REQ_LINE_VALVE_2 := "LTLP_DirectKeyGetMovNoData".PowerUp[4], HMI_REQ_LINE_VALVE_3 := "LTLP_DirectKeyGetMovNoData".PowerUp[5], HMI_REQ_LINE_VALVE_4 :=, HMI_POWER_UP_COND_OFF_VALVE_1 => "LTLP_HMIProInterfaceData".powerupCondOff3, HMI_POWER_UP_COND_ON_VALVE_1 => "LTLP_HMIProInterfaceData".powerupCondOn3, HMI_POWER_UP_EXECU_LEFT_VALVE_1 => "LTLP_HMIProInterfaceData".powerup3ExecutableLeft, HMI_POWER_UP_EXECU_RIGHT_VALVE_1 => "LTLP_HMIProInterfaceData".powerup3ExecutableRight, HMI_POWER_UP_COND_OFF_VALVE_2 => "LTLP_HMIProInterfaceData".powerupCondOff4, HMI_POWER_UP_COND_ON_VALVE_2 => "LTLP_HMIProInterfaceData".powerupCondOn4, HMI_POWER_UP_EXECU_LEFT_VALVE_2 => "LTLP_HMIProInterfaceData".powerup4ExecutableLeft, HMI_POWER_UP_EXECU_RIGHT_VALVE_2 => "LTLP_HMIProInterfaceData".powerup4ExecutableRight, HMI_POWER_UP_COND_OFF_VALVE_3 => "LTLP_HMIProInterfaceData".powerupCondOff5, HMI_POWER_UP_COND_ON_VALVE_3 => "LTLP_HMIProInterfaceData".powerupCondOn5, HMI_POWER_UP_EXECU_LEFT_VALVE_3 => "LTLP_HMIProInterfaceData".powerup5ExecutableLeft, HMI_POWER_UP_EXECU_RIGHT_VALVE_3 => "LTLP_HMIProInterfaceData".powerup5ExecutableRight, HMI_POWER_UP_COND_OFF_VALVE_4 =>, HMI_POWER_UP_COND_ON_VALVE_4 =>, HMI_POWER_UP_EXECU_LEFT_VALVE_4 =>, HMI_POWER_UP_EXECU_RIGHT_VALVE_4 =>, MOTOR => "LB_PMP_ON_Q", VALVE_1 => "LB_VLV_1_ON_Q", VALVE_2 => "LB_VLV_2_ON_Q", VALVE_3 => "LB_VLV_3_ON_Q", VALVE_4 =>)
   END_RUNG
   // the same network as SCL:
   "DB1421_PROGRESSIVE_LUBRICATION_WITH_GREASE"(OPTIONS_0 := 2#1010_0000,   // "FB1403_PROGRESSIVE_LUBRICATION_WITH_GREASE"
                           OPTIONS_1 := 2#0000_0011,
                           TIME_VALVE_1 := T#5d,
                           TIME_VALVE_3 := T#5d,
                           PULSES_PER_CYCLE_VALVE_1 := 2,
                           PULSES_PER_CYCLE_VALVE_2 := 2,
                           PULSES_PER_CYCLE_VALVE_3 := 2,
                           PULSES_PER_CYCLE_VALVE_4 := 2,
                           LUBRICATION_DONE_1 := "LB_BRANCH_1_DONE",
                           LUBRICATION_DONE_2 := "LB_BRANCH_2_DONE",
                           LUBRICATION_DONE_3 := "LB_BRANCH_3_DONE",
                           SWITCH_ON_VALVE_1_DIST_REQ_AXIS_1 := "LBP_Axis12".E_ScratchPulse,
                           SWITCH_ON_VALVE_1_DIST_REQ_AXIS_2 := "LBP_Axis26".E_ScratchPulse,
                           SWITCH_ON_VALVE_2_DIST_REQ_AXIS_1 := "LBP_Axis8".E_ScratchPulse,
                           SWITCH_ON_VALVE_2_DIST_REQ_AXIS_2 := "LBP_Axis22".E_ScratchPulse,
                           HMI_REQ_LINE_VALVE_1 := "LTLP_DirectKeyGetMovNoData".PowerUp[3],
                           HMI_REQ_LINE_VALVE_2 := "LTLP_DirectKeyGetMovNoData".PowerUp[4],
                           HMI_REQ_LINE_VALVE_3 := "LTLP_DirectKeyGetMovNoData".PowerUp[5],
                           HMI_POWER_UP_COND_OFF_VALVE_1 => "LTLP_HMIProInterfaceData".powerupCondOff3,
                           HMI_POWER_UP_COND_ON_VALVE_1 => "LTLP_HMIProInterfaceData".powerupCondOn3,
                           HMI_POWER_UP_EXECU_LEFT_VALVE_1 => "LTLP_HMIProInterfaceData".powerup3ExecutableLeft,
                           HMI_POWER_UP_EXECU_RIGHT_VALVE_1 => "LTLP_HMIProInterfaceData".powerup3ExecutableRight,
                           HMI_POWER_UP_COND_OFF_VALVE_2 => "LTLP_HMIProInterfaceData".powerupCondOff4,
                           HMI_POWER_UP_COND_ON_VALVE_2 => "LTLP_HMIProInterfaceData".powerupCondOn4,
                           HMI_POWER_UP_EXECU_LEFT_VALVE_2 => "LTLP_HMIProInterfaceData".powerup4ExecutableLeft,
                           HMI_POWER_UP_EXECU_RIGHT_VALVE_2 => "LTLP_HMIProInterfaceData".powerup4ExecutableRight,
                           HMI_POWER_UP_COND_OFF_VALVE_3 => "LTLP_HMIProInterfaceData".powerupCondOff5,
                           HMI_POWER_UP_COND_ON_VALVE_3 => "LTLP_HMIProInterfaceData".powerupCondOn5,
                           HMI_POWER_UP_EXECU_LEFT_VALVE_3 => "LTLP_HMIProInterfaceData".powerup5ExecutableLeft,
                           HMI_POWER_UP_EXECU_RIGHT_VALVE_3 => "LTLP_HMIProInterfaceData".powerup5ExecutableRight,
                           MOTOR => "LB_PMP_ON_Q",
                           VALVE_1 => "LB_VLV_1_ON_Q",
                           VALVE_2 => "LB_VLV_2_ON_Q",
                           VALVE_3 => "LB_VLV_3_ON_Q");
END_REGION

REGION Network 5: <<<<<<<<<<<<<<<<<<<< GENERAL WARNINGS >>>>>>>>>>>>>>>>>>>>
END_REGION

REGION Network 6: (WRN) SELECT AUTO OR SEMI MODE TO POWER ON SERVICES
   RUNG wire#powerrail
      Contact( "DB1401_PNEUMATIC_SYSTEM".IN_SERVICE )
      Not()
      Contact( "DB2001_MODES_GENERAL".MG1.GENERAL.MANUAL_SELECTED )
      Contact( "DB2120_MPP_ITC_IPC".START_SERVICES_GLOBAL )
      S_Coil( "DB426_ALARMS_WARNINGS".ALARMS.WARNINGS."740077" )
   END_RUNG
   // the same network as SCL:
   IF NOT "DB1401_PNEUMATIC_SYSTEM".IN_SERVICE AND "DB2001_MODES_GENERAL".MG1.GENERAL.MANUAL_SELECTED AND "DB2120_MPP_ITC_IPC".START_SERVICES_GLOBAL THEN
       "DB426_ALARMS_WARNINGS".ALARMS.WARNINGS."740077" := TRUE;
   END_IF;
END_REGION

REGION Network 7: (WRN) SELECT AUTO OR SEMI MODE TO POWER ON SERVICES
   RUNG wire#powerrail
      Contact( "DB1401_PNEUMATIC_SYSTEM".IN_SERVICE )
      wire#w1
      R_Coil( "DB426_ALARMS_WARNINGS".ALARMS.WARNINGS."740077" )
   END_RUNG
   RUNG wire#powerrail
      Contact( "DB2120_MPP_ITC_IPC".RESET_FAULTS )
   END_RUNG wire#w1
   // the same network as SCL:
   IF "DB1401_PNEUMATIC_SYSTEM".IN_SERVICE OR "DB2120_MPP_ITC_IPC".RESET_FAULTS THEN
       "DB426_ALARMS_WARNINGS".ALARMS.WARNINGS."740077" := FALSE;
   END_IF;
END_REGION

REGION Network 8: WARNINGS
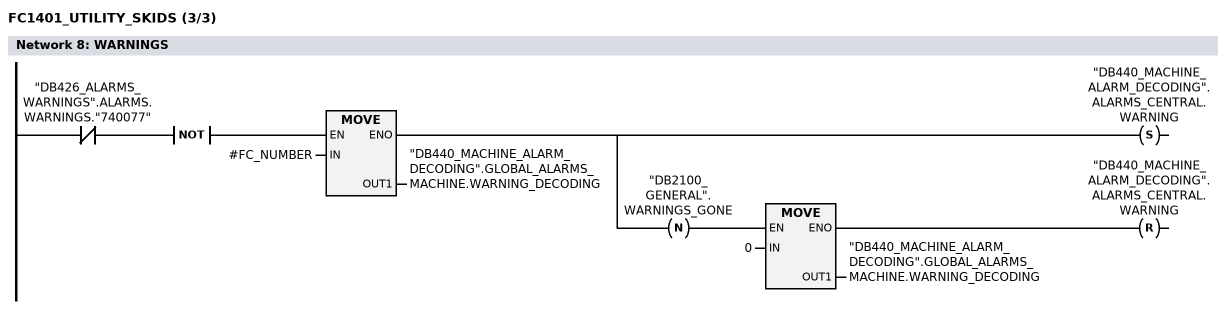
   RUNG wire#powerrail
      I_Contact( "DB426_ALARMS_WARNINGS".ALARMS.WARNINGS."740077" )
      Not()
      { S7_GenerateENO := "TRUE" } Move(in := #FC_NUMBER, out1 => "DB440_MACHINE_ALARM_DECODING".GLOBAL_ALARMS_MACHINE.WARNING_DECODING)
      wire#w1
      S_Coil( "DB440_MACHINE_ALARM_DECODING".ALARMS_CENTRAL.WARNING )
   END_RUNG
   RUNG wire#w1
      N_Trig( "DB2100_GENERAL".WARNINGS_GONE )
      { S7_GenerateENO := "TRUE" } Move(in := 0, out1 => "DB440_MACHINE_ALARM_DECODING".GLOBAL_ALARMS_MACHINE.WARNING_DECODING)
      R_Coil( "DB440_MACHINE_ALARM_DECODING".ALARMS_CENTRAL.WARNING )
   END_RUNG
   // the same network as SCL:
   // ENO of a box is taken as its EN; it also drops when the box reports an error
   #_w1 := NOT (NOT "DB426_ALARMS_WARNINGS".ALARMS.WARNINGS."740077");
   IF #_w1 THEN
       "DB440_MACHINE_ALARM_DECODING".GLOBAL_ALARMS_MACHINE.WARNING_DECODING := #FC_NUMBER;
       "DB440_MACHINE_ALARM_DECODING".ALARMS_CENTRAL.WARNING := TRUE;
   END_IF;
   #_w2 := NOT #_w1 AND "DB2100_GENERAL".WARNINGS_GONE;   // falling edge
   "DB2100_GENERAL".WARNINGS_GONE := #_w1;
   IF #_w2 THEN
       "DB440_MACHINE_ALARM_DECODING".GLOBAL_ALARMS_MACHINE.WARNING_DECODING := 0;
       "DB440_MACHINE_ALARM_DECODING".ALARMS_CENTRAL.WARNING := FALSE;
   END_IF;
END_REGION
END_FUNCTION

FUNCTION "FC1450_COOLING_GENERAL" : Void   // FC1450, LAD
{ S7_Optimized_Access := 'TRUE' }
VERSION : 0.1
// stored: AutoNumber false, IsIECCheckEnabled false, SetENOAutomatically false, UDAEnableTagReadback false
BEGIN

REGION Network 1: CALL FC1451_MACHINE_MAIN_COOLING_SYSTEM
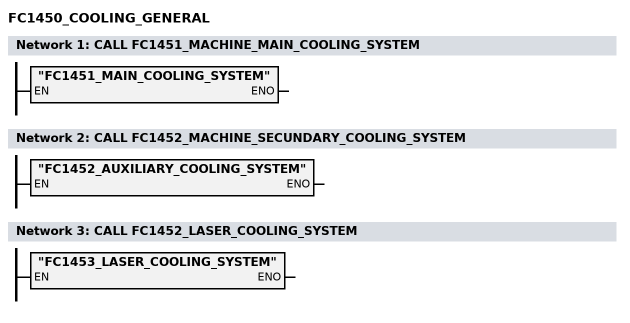
   RUNG wire#powerrail
      "FC1451_MAIN_COOLING_SYSTEM"()
   END_RUNG
   // the same network as SCL:
   "FC1451_MAIN_COOLING_SYSTEM"();
END_REGION

REGION Network 2: CALL FC1452_MACHINE_SECUNDARY_COOLING_SYSTEM
   RUNG wire#powerrail
      "FC1452_AUXILIARY_COOLING_SYSTEM"()
   END_RUNG
   // the same network as SCL:
   "FC1452_AUXILIARY_COOLING_SYSTEM"();
END_REGION

REGION Network 3: CALL FC1452_LASER_COOLING_SYSTEM
   RUNG wire#powerrail
      "FC1453_LASER_COOLING_SYSTEM"()
   END_RUNG
   // the same network as SCL:
   "FC1453_LASER_COOLING_SYSTEM"();
END_REGION
END_FUNCTION

FUNCTION "FC1500_GAS_GENERAL" : Void   // FC1500, LAD
{ S7_Optimized_Access := 'TRUE' }
VERSION : 0.1
// stored: AutoNumber false, IsIECCheckEnabled false, SetENOAutomatically false, UDAEnableTagReadback false
BEGIN

REGION Network 1: CALL FC1501_MAIN_GAS_VALVE
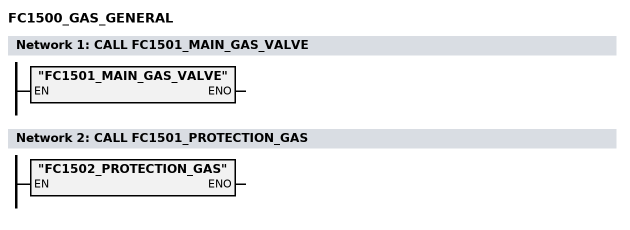
   RUNG wire#powerrail
      "FC1501_MAIN_GAS_VALVE"()
   END_RUNG
   // the same network as SCL:
   "FC1501_MAIN_GAS_VALVE"();
END_REGION

REGION Network 2: CALL FC1501_PROTECTION_GAS
   RUNG wire#powerrail
      "FC1502_PROTECTION_GAS"()
   END_RUNG
   // the same network as SCL:
   "FC1502_PROTECTION_GAS"();
END_REGION
END_FUNCTION

FUNCTION "FC1700_ASPIRATION_GENERAL" : Void   // FC1700, LAD
{ S7_Optimized_Access := 'FALSE' }
AUTHOR : ETXETAR
VERSION : 1.0
// stored: AutoNumber false, IsIECCheckEnabled false, SetENOAutomatically false, UDAEnableTagReadback false
   VAR CONSTANT
      FC_NUMBER : DInt := 1700;
   END_VAR
BEGIN

REGION Network 1: CALL FC1701_KELLER_ASPIRATION_CONTROL
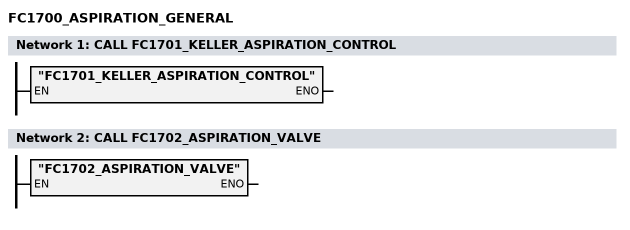
   RUNG wire#powerrail
      "FC1701_KELLER_ASPIRATION_CONTROL"()
   END_RUNG
   // the same network as SCL:
   "FC1701_KELLER_ASPIRATION_CONTROL"();
END_REGION

REGION Network 2: CALL FC1702_ASPIRATION_VALVE
   RUNG wire#powerrail
      "FC1702_ASPIRATION_VALVE"()
   END_RUNG
   // the same network as SCL:
   "FC1702_ASPIRATION_VALVE"();
END_REGION
END_FUNCTION

FUNCTION "FC1800_CLEANING_VALVES_GENERAL" : Void   // FC1800, LAD
{ S7_Optimized_Access := 'TRUE' }
VERSION : 0.1
// stored: AutoNumber false, IsIECCheckEnabled false, SetENOAutomatically false, UDAEnableTagReadback false
BEGIN

REGION Network 1: <<<<<<<<<<<<<<<<<<<< CLEANING VALVES >>>>>>>>>>>>>>>>>>>>
END_REGION

REGION Network 2: UNIT 01CLEANING VALVE
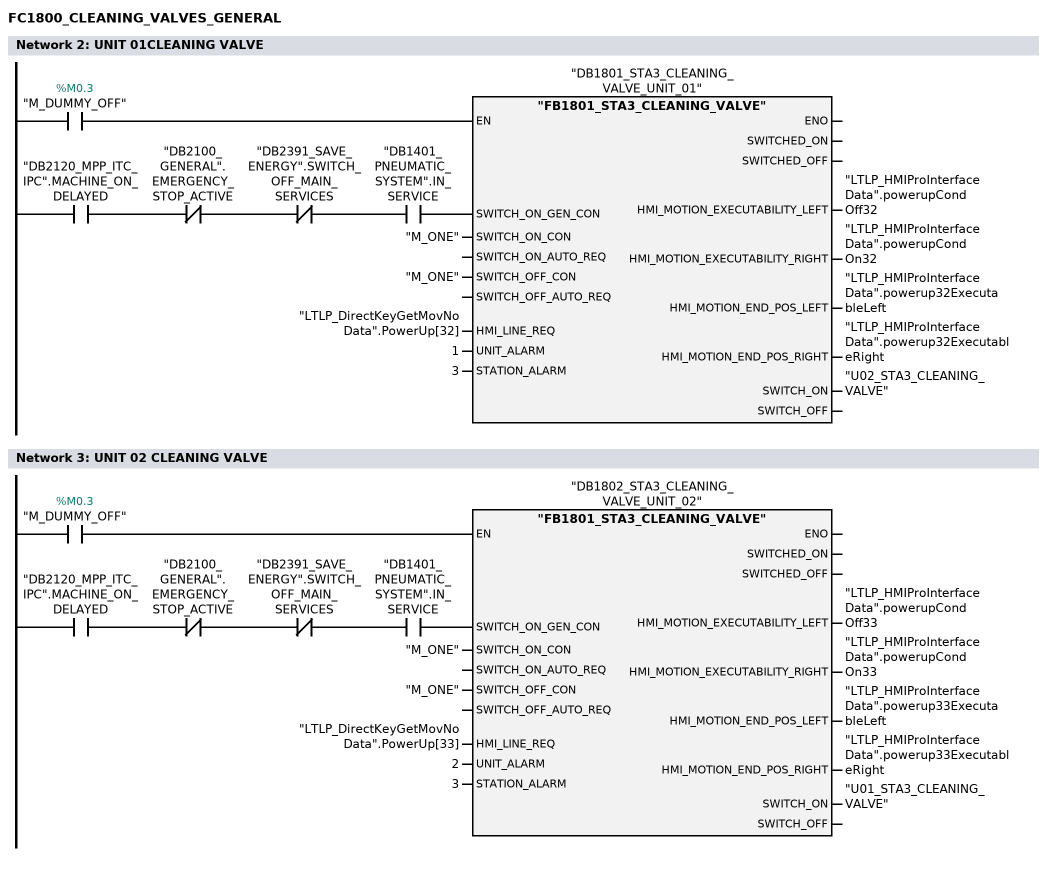
   RUNG wire#powerrail
      Contact( "M_DUMMY_OFF" )
      "DB1801_STA3_CLEANING_VALVE_UNIT_01"(SWITCH_ON_GEN_CON := wire#w1, SWITCH_ON_CON := "M_ONE", SWITCH_ON_AUTO_REQ :=, SWITCH_OFF_CON := "M_ONE", SWITCH_OFF_AUTO_REQ :=, HMI_LINE_REQ := "LTLP_DirectKeyGetMovNoData".PowerUp[32], UNIT_ALARM := 1, STATION_ALARM := 3, SWITCHED_ON =>, SWITCHED_OFF =>, HMI_MOTION_EXECUTABILITY_LEFT => "LTLP_HMIProInterfaceData".powerupCondOff32, HMI_MOTION_EXECUTABILITY_RIGHT => "LTLP_HMIProInterfaceData".powerupCondOn32, HMI_MOTION_END_POS_LEFT => "LTLP_HMIProInterfaceData".powerup32ExecutableLeft, HMI_MOTION_END_POS_RIGHT => "LTLP_HMIProInterfaceData".powerup32ExecutableRight, SWITCH_ON => "U02_STA3_CLEANING_VALVE", SWITCH_OFF =>)
   END_RUNG
   RUNG wire#powerrail
      Contact( "DB2120_MPP_ITC_IPC".MACHINE_ON_DELAYED )
      I_Contact( "DB2100_GENERAL".EMERGENCY_STOP_ACTIVE )
      I_Contact( "DB2391_SAVE_ENERGY".SWITCH_OFF_MAIN_SERVICES )
      Contact( "DB1401_PNEUMATIC_SYSTEM".IN_SERVICE )
   END_RUNG wire#w1
   // the same network as SCL:
   IF "M_DUMMY_OFF" THEN
       "DB1801_STA3_CLEANING_VALVE_UNIT_01"(SWITCH_ON_GEN_CON := "DB2120_MPP_ITC_IPC".MACHINE_ON_DELAYED AND NOT "DB2100_GENERAL".EMERGENCY_STOP_ACTIVE AND NOT "DB2391_SAVE_ENERGY".SWITCH_OFF_MAIN_SERVICES AND "DB1401_PNEUMATIC_SYSTEM".IN_SERVICE,   // "FB1801_STA3_CLEANING_VALVE"
                               SWITCH_ON_CON := "M_ONE",
                               SWITCH_OFF_CON := "M_ONE",
                               HMI_LINE_REQ := "LTLP_DirectKeyGetMovNoData".PowerUp[32],
                               UNIT_ALARM := 1,
                               STATION_ALARM := 3,
                               HMI_MOTION_EXECUTABILITY_LEFT => "LTLP_HMIProInterfaceData".powerupCondOff32,
                               HMI_MOTION_EXECUTABILITY_RIGHT => "LTLP_HMIProInterfaceData".powerupCondOn32,
                               HMI_MOTION_END_POS_LEFT => "LTLP_HMIProInterfaceData".powerup32ExecutableLeft,
                               HMI_MOTION_END_POS_RIGHT => "LTLP_HMIProInterfaceData".powerup32ExecutableRight,
                               SWITCH_ON => "U02_STA3_CLEANING_VALVE");
   END_IF;
END_REGION

REGION Network 3: UNIT 02 CLEANING VALVE
   RUNG wire#powerrail
      Contact( "M_DUMMY_OFF" )
      "DB1802_STA3_CLEANING_VALVE_UNIT_02"(SWITCH_ON_GEN_CON := wire#w1, SWITCH_ON_CON := "M_ONE", SWITCH_ON_AUTO_REQ :=, SWITCH_OFF_CON := "M_ONE", SWITCH_OFF_AUTO_REQ :=, HMI_LINE_REQ := "LTLP_DirectKeyGetMovNoData".PowerUp[33], UNIT_ALARM := 2, STATION_ALARM := 3, SWITCHED_ON =>, SWITCHED_OFF =>, HMI_MOTION_EXECUTABILITY_LEFT => "LTLP_HMIProInterfaceData".powerupCondOff33, HMI_MOTION_EXECUTABILITY_RIGHT => "LTLP_HMIProInterfaceData".powerupCondOn33, HMI_MOTION_END_POS_LEFT => "LTLP_HMIProInterfaceData".powerup33ExecutableLeft, HMI_MOTION_END_POS_RIGHT => "LTLP_HMIProInterfaceData".powerup33ExecutableRight, SWITCH_ON => "U01_STA3_CLEANING_VALVE", SWITCH_OFF =>)
   END_RUNG
   RUNG wire#powerrail
      Contact( "DB2120_MPP_ITC_IPC".MACHINE_ON_DELAYED )
      I_Contact( "DB2100_GENERAL".EMERGENCY_STOP_ACTIVE )
      I_Contact( "DB2391_SAVE_ENERGY".SWITCH_OFF_MAIN_SERVICES )
      Contact( "DB1401_PNEUMATIC_SYSTEM".IN_SERVICE )
   END_RUNG wire#w1
   // the same network as SCL:
   IF "M_DUMMY_OFF" THEN
       "DB1802_STA3_CLEANING_VALVE_UNIT_02"(SWITCH_ON_GEN_CON := "DB2120_MPP_ITC_IPC".MACHINE_ON_DELAYED AND NOT "DB2100_GENERAL".EMERGENCY_STOP_ACTIVE AND NOT "DB2391_SAVE_ENERGY".SWITCH_OFF_MAIN_SERVICES AND "DB1401_PNEUMATIC_SYSTEM".IN_SERVICE,   // "FB1801_STA3_CLEANING_VALVE"
                               SWITCH_ON_CON := "M_ONE",
                               SWITCH_OFF_CON := "M_ONE",
                               HMI_LINE_REQ := "LTLP_DirectKeyGetMovNoData".PowerUp[33],
                               UNIT_ALARM := 2,
                               STATION_ALARM := 3,
                               HMI_MOTION_EXECUTABILITY_LEFT => "LTLP_HMIProInterfaceData".powerupCondOff33,
                               HMI_MOTION_EXECUTABILITY_RIGHT => "LTLP_HMIProInterfaceData".powerupCondOn33,
                               HMI_MOTION_END_POS_LEFT => "LTLP_HMIProInterfaceData".powerup33ExecutableLeft,
                               HMI_MOTION_END_POS_RIGHT => "LTLP_HMIProInterfaceData".powerup33ExecutableRight,
                               SWITCH_ON => "U01_STA3_CLEANING_VALVE");
   END_IF;
END_REGION
END_FUNCTION

FUNCTION "FC2000_MACHINE_MODES" : Void   // FC2000, LAD
{ S7_Optimized_Access := 'FALSE' }
AUTHOR : ETXETAR
VERSION : 1.0
// stored: AutoNumber false, IsIECCheckEnabled false, SetENOAutomatically false, UDAEnableTagReadback false
BEGIN

REGION Network 1: OPTIONS OFF
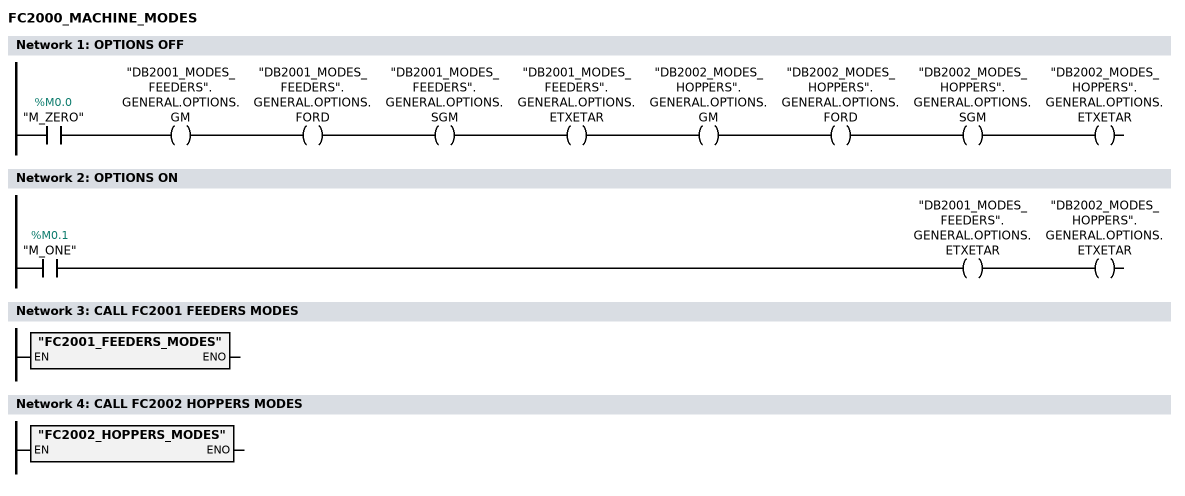
   RUNG wire#powerrail
      Contact( "M_ZERO" )
      Coil( "DB2001_MODES_FEEDERS".GENERAL.OPTIONS.GM )
      Coil( "DB2001_MODES_FEEDERS".GENERAL.OPTIONS.FORD )
      Coil( "DB2001_MODES_FEEDERS".GENERAL.OPTIONS.SGM )
      Coil( "DB2001_MODES_FEEDERS".GENERAL.OPTIONS.ETXETAR )
      Coil( "DB2002_MODES_HOPPERS".GENERAL.OPTIONS.GM )
      Coil( "DB2002_MODES_HOPPERS".GENERAL.OPTIONS.FORD )
      Coil( "DB2002_MODES_HOPPERS".GENERAL.OPTIONS.SGM )
      Coil( "DB2002_MODES_HOPPERS".GENERAL.OPTIONS.ETXETAR )
   END_RUNG
   // the same network as SCL:
   "DB2001_MODES_FEEDERS".GENERAL.OPTIONS.GM := "M_ZERO";
   "DB2001_MODES_FEEDERS".GENERAL.OPTIONS.FORD := "M_ZERO";
   "DB2001_MODES_FEEDERS".GENERAL.OPTIONS.SGM := "M_ZERO";
   "DB2001_MODES_FEEDERS".GENERAL.OPTIONS.ETXETAR := "M_ZERO";
   "DB2002_MODES_HOPPERS".GENERAL.OPTIONS.GM := "M_ZERO";
   "DB2002_MODES_HOPPERS".GENERAL.OPTIONS.FORD := "M_ZERO";
   "DB2002_MODES_HOPPERS".GENERAL.OPTIONS.SGM := "M_ZERO";
   "DB2002_MODES_HOPPERS".GENERAL.OPTIONS.ETXETAR := "M_ZERO";
END_REGION

REGION Network 2: OPTIONS ON
   RUNG wire#powerrail
      Contact( "M_ONE" )
      Coil( "DB2001_MODES_FEEDERS".GENERAL.OPTIONS.ETXETAR )
      Coil( "DB2002_MODES_HOPPERS".GENERAL.OPTIONS.ETXETAR )
   END_RUNG
   // the same network as SCL:
   "DB2001_MODES_FEEDERS".GENERAL.OPTIONS.ETXETAR := "M_ONE";
   "DB2002_MODES_HOPPERS".GENERAL.OPTIONS.ETXETAR := "M_ONE";
END_REGION

REGION Network 3: CALL FC2001 FEEDERS MODES
   RUNG wire#powerrail
      "FC2001_FEEDERS_MODES"()
   END_RUNG
   // the same network as SCL:
   "FC2001_FEEDERS_MODES"();
END_REGION

REGION Network 4: CALL FC2002 HOPPERS MODES
   RUNG wire#powerrail
      "FC2002_HOPPERS_MODES"()
   END_RUNG
   // the same network as SCL:
   "FC2002_HOPPERS_MODES"();
END_REGION
END_FUNCTION

FUNCTION "FC2030_MACHINE_CYCLES" : Void   // FC2030, LAD
{ S7_Optimized_Access := 'FALSE' }
AUTHOR : ETXETAR
VERSION : 1.0
// stored: AutoNumber false, IsIECCheckEnabled false, SetENOAutomatically false, UDAEnableTagReadback false
BEGIN

REGION Network 1: CALL FC2031 MACHINE CONTINUOUS CYCLE
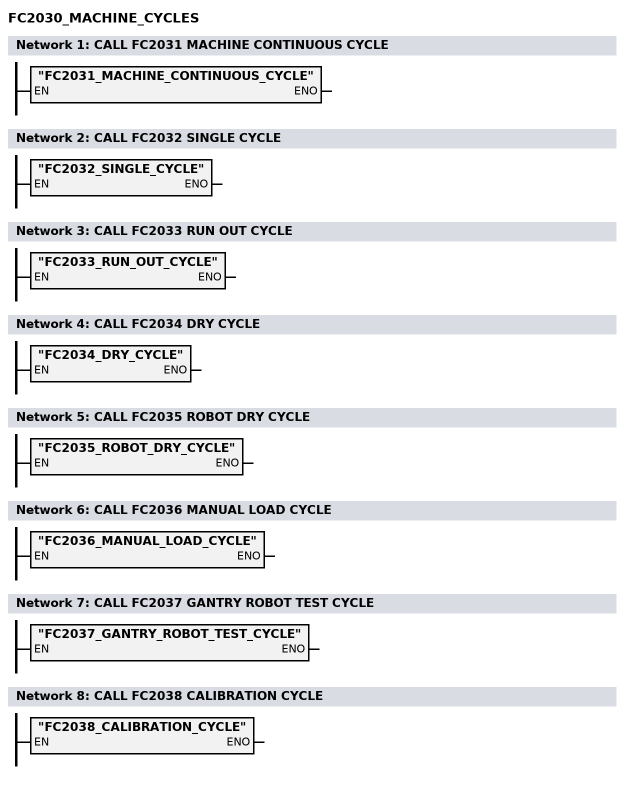
   RUNG wire#powerrail
      "FC2031_MACHINE_CONTINUOUS_CYCLE"()
   END_RUNG
   // the same network as SCL:
   "FC2031_MACHINE_CONTINUOUS_CYCLE"();
END_REGION

REGION Network 2: CALL FC2032 SINGLE CYCLE
   RUNG wire#powerrail
      "FC2032_SINGLE_CYCLE"()
   END_RUNG
   // the same network as SCL:
   "FC2032_SINGLE_CYCLE"();
END_REGION

REGION Network 3: CALL FC2033 RUN OUT CYCLE
   RUNG wire#powerrail
      "FC2033_RUN_OUT_CYCLE"()
   END_RUNG
   // the same network as SCL:
   "FC2033_RUN_OUT_CYCLE"();
END_REGION

REGION Network 4: CALL FC2034 DRY CYCLE
   RUNG wire#powerrail
      "FC2034_DRY_CYCLE"()
   END_RUNG
   // the same network as SCL:
   "FC2034_DRY_CYCLE"();
END_REGION

REGION Network 5: CALL FC2035 ROBOT DRY CYCLE
   RUNG wire#powerrail
      "FC2035_ROBOT_DRY_CYCLE"()
   END_RUNG
   // the same network as SCL:
   "FC2035_ROBOT_DRY_CYCLE"();
END_REGION

REGION Network 6: CALL FC2036 MANUAL LOAD CYCLE
   RUNG wire#powerrail
      "FC2036_MANUAL_LOAD_CYCLE"()
   END_RUNG
   // the same network as SCL:
   "FC2036_MANUAL_LOAD_CYCLE"();
END_REGION

REGION Network 7: CALL FC2037 GANTRY ROBOT TEST CYCLE
   RUNG wire#powerrail
      "FC2037_GANTRY_ROBOT_TEST_CYCLE"()
   END_RUNG
   // the same network as SCL:
   "FC2037_GANTRY_ROBOT_TEST_CYCLE"();
END_REGION

REGION Network 8: CALL FC2038 CALIBRATION CYCLE
   RUNG wire#powerrail
      "FC2038_CALIBRATION_CYCLE"()
   END_RUNG
   // the same network as SCL:
   "FC2038_CALIBRATION_CYCLE"();
END_REGION
END_FUNCTION

FUNCTION "FC2100_GENERAL" : Void   // FC2100, LAD
{ S7_Optimized_Access := 'FALSE' }
AUTHOR : ETXETAR
VERSION : 1.0
// stored: AutoNumber false, IsIECCheckEnabled false, SetENOAutomatically false, UDAEnableTagReadback false
   VAR CONSTANT
      FC_NUMBER : DInt := 2100;   // FC NUMBER
   END_VAR
BEGIN

REGION Network 1: ALWAYS OFF
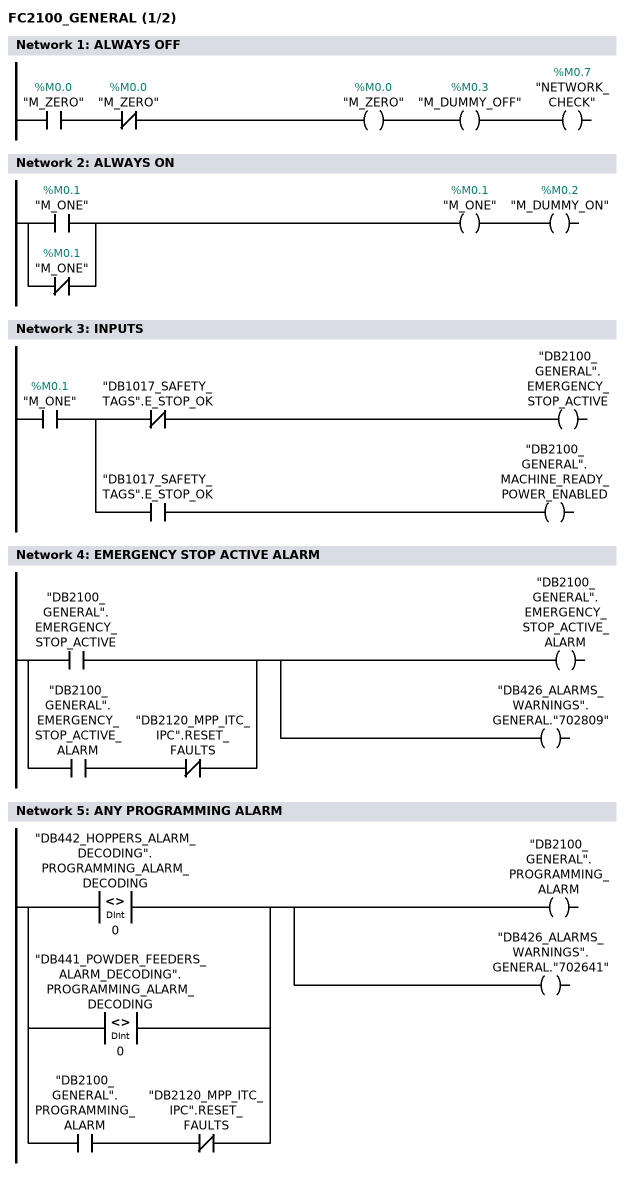
   RUNG wire#powerrail
      Contact( "M_ZERO" )
      I_Contact( "M_ZERO" )
      Coil( "M_ZERO" )
      Coil( "M_DUMMY_OFF" )
      Coil( "NETWORK_CHECK" )
   END_RUNG
   // the same network as SCL:
   "M_ZERO" := "M_ZERO" AND NOT "M_ZERO";
   "M_DUMMY_OFF" := "M_ZERO";
   "NETWORK_CHECK" := "M_ZERO";
END_REGION

REGION Network 2: ALWAYS ON
   RUNG wire#powerrail
      Contact( "M_ONE" )
      wire#w1
      Coil( "M_ONE" )
      Coil( "M_DUMMY_ON" )
   END_RUNG
   RUNG wire#powerrail
      I_Contact( "M_ONE" )
   END_RUNG wire#w1
   // the same network as SCL:
   "M_ONE" := "M_ONE" OR NOT "M_ONE";
   "M_DUMMY_ON" := "M_ONE";
END_REGION

REGION Network 3: INPUTS
   RUNG wire#powerrail
      Contact( "M_ONE" )
      wire#w1
      I_Contact( "DB1017_SAFETY_TAGS".E_STOP_OK )
      Coil( "DB2100_GENERAL".EMERGENCY_STOP_ACTIVE )
   END_RUNG
   RUNG wire#w1
      Contact( "DB1017_SAFETY_TAGS".E_STOP_OK )
      Coil( "DB2100_GENERAL".MACHINE_READY_POWER_ENABLED )
   END_RUNG
   // the same network as SCL:
   "DB2100_GENERAL".EMERGENCY_STOP_ACTIVE := "M_ONE" AND NOT "DB1017_SAFETY_TAGS".E_STOP_OK;
   "DB2100_GENERAL".MACHINE_READY_POWER_ENABLED := "M_ONE" AND "DB1017_SAFETY_TAGS".E_STOP_OK;
END_REGION

REGION Network 4: EMERGENCY STOP ACTIVE ALARM
   RUNG wire#powerrail
      Contact( "DB2100_GENERAL".EMERGENCY_STOP_ACTIVE )
      wire#w1
      Coil( "DB2100_GENERAL".EMERGENCY_STOP_ACTIVE_ALARM )
   END_RUNG
   RUNG wire#powerrail
      Contact( "DB2100_GENERAL".EMERGENCY_STOP_ACTIVE_ALARM )
      I_Contact( "DB2120_MPP_ITC_IPC".RESET_FAULTS )
   END_RUNG wire#w1
   RUNG wire#w1
      Coil( "DB426_ALARMS_WARNINGS".GENERAL."702809" )
   END_RUNG
   // the same network as SCL:
   "DB2100_GENERAL".EMERGENCY_STOP_ACTIVE_ALARM := "DB2100_GENERAL".EMERGENCY_STOP_ACTIVE OR ("DB2100_GENERAL".EMERGENCY_STOP_ACTIVE_ALARM AND NOT "DB2120_MPP_ITC_IPC".RESET_FAULTS);
   "DB426_ALARMS_WARNINGS".GENERAL."702809" := "DB2100_GENERAL".EMERGENCY_STOP_ACTIVE_ALARM;
END_REGION

REGION Network 5: ANY PROGRAMMING ALARM
   RUNG wire#powerrail
      { S7_Templates := "SrcType := DInt" } NE_Contact(in1 := "DB442_HOPPERS_ALARM_DECODING".PROGRAMMING_ALARM_DECODING, in2 := 0)
      wire#w1
      Coil( "DB2100_GENERAL".PROGRAMMING_ALARM )
   END_RUNG
   RUNG wire#powerrail
      { S7_Templates := "SrcType := DInt" } NE_Contact(in1 := "DB441_POWDER_FEEDERS_ALARM_DECODING".PROGRAMMING_ALARM_DECODING, in2 := 0)
   END_RUNG wire#w1
   RUNG wire#powerrail
      Contact( "DB2100_GENERAL".PROGRAMMING_ALARM )
      I_Contact( "DB2120_MPP_ITC_IPC".RESET_FAULTS )
   END_RUNG wire#w1
   RUNG wire#w1
      Coil( "DB426_ALARMS_WARNINGS".GENERAL."702641" )
   END_RUNG
   // the same network as SCL:
   "DB2100_GENERAL".PROGRAMMING_ALARM := ("DB442_HOPPERS_ALARM_DECODING".PROGRAMMING_ALARM_DECODING <> 0) OR ("DB441_POWDER_FEEDERS_ALARM_DECODING".PROGRAMMING_ALARM_DECODING <> 0) OR ("DB2100_GENERAL".PROGRAMMING_ALARM AND NOT "DB2120_MPP_ITC_IPC".RESET_FAULTS);
   "DB426_ALARMS_WARNINGS".GENERAL."702641" := "DB2100_GENERAL".PROGRAMMING_ALARM;
END_REGION

REGION Network 6: CHECK NETWORK LOGIC ALARM
   // CHECK EVERY NETWORK LOGIC WHERE THE M0.7 IS PROGRAMMED, THOSE NETWORK MUST BE ADAPTED ACCORDING TO THE MACHINE STRUCTURE
   // 
   // DELETE THIS NETWORK
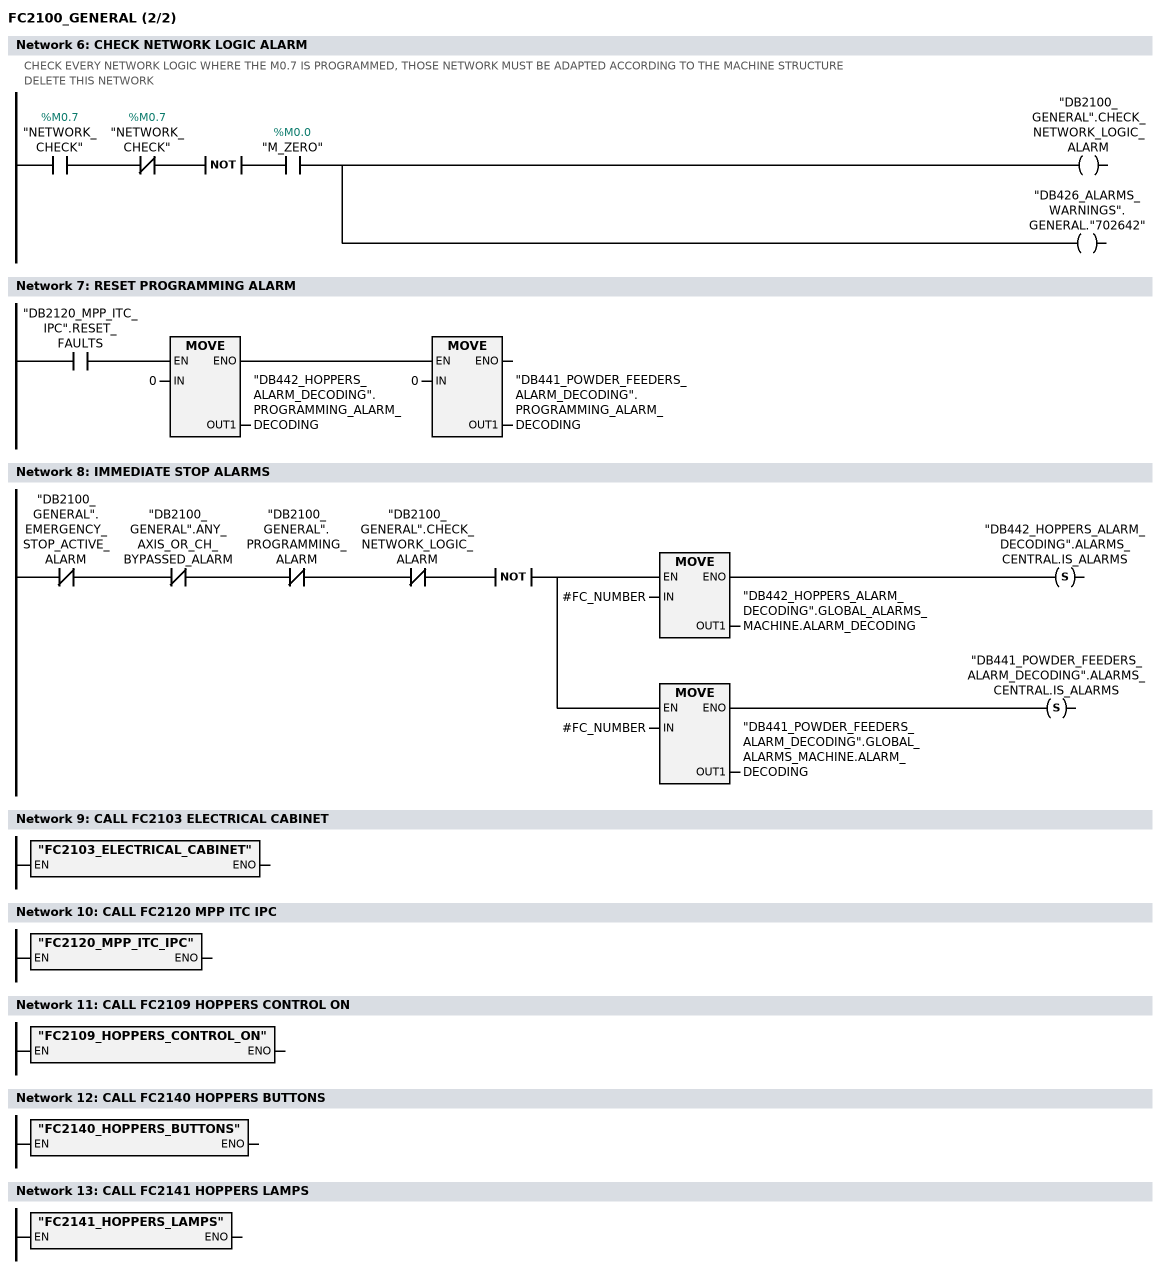
   RUNG wire#powerrail
      Contact( "NETWORK_CHECK" )
      I_Contact( "NETWORK_CHECK" )
      Not()
      Contact( "M_ZERO" )
      wire#w1
      Coil( "DB2100_GENERAL".CHECK_NETWORK_LOGIC_ALARM )
   END_RUNG
   RUNG wire#w1
      Coil( "DB426_ALARMS_WARNINGS".GENERAL."702642" )
   END_RUNG
   // the same network as SCL:
   "DB2100_GENERAL".CHECK_NETWORK_LOGIC_ALARM := NOT ("NETWORK_CHECK" AND NOT "NETWORK_CHECK") AND "M_ZERO";
   "DB426_ALARMS_WARNINGS".GENERAL."702642" := "DB2100_GENERAL".CHECK_NETWORK_LOGIC_ALARM;
END_REGION

REGION Network 7: RESET PROGRAMMING ALARM
   RUNG wire#powerrail
      Contact( "DB2120_MPP_ITC_IPC".RESET_FAULTS )
      { S7_GenerateENO := "TRUE" } Move(in := 0, out1 => "DB442_HOPPERS_ALARM_DECODING".PROGRAMMING_ALARM_DECODING)
      { S7_GenerateENO := "TRUE" } Move(in := 0, out1 => "DB441_POWDER_FEEDERS_ALARM_DECODING".PROGRAMMING_ALARM_DECODING)
   END_RUNG
   // the same network as SCL:
   // ENO of a box is taken as its EN; it also drops when the box reports an error
   IF "DB2120_MPP_ITC_IPC".RESET_FAULTS THEN
       "DB442_HOPPERS_ALARM_DECODING".PROGRAMMING_ALARM_DECODING := 0;
       "DB441_POWDER_FEEDERS_ALARM_DECODING".PROGRAMMING_ALARM_DECODING := 0;
   END_IF;
END_REGION

REGION Network 8: IMMEDIATE STOP ALARMS
   RUNG wire#powerrail
      I_Contact( "DB2100_GENERAL".EMERGENCY_STOP_ACTIVE_ALARM )
      I_Contact( "DB2100_GENERAL".ANY_AXIS_OR_CH_BYPASSED_ALARM )
      I_Contact( "DB2100_GENERAL".PROGRAMMING_ALARM )
      I_Contact( "DB2100_GENERAL".CHECK_NETWORK_LOGIC_ALARM )
      Not()
      wire#w1
      { S7_GenerateENO := "TRUE" } Move(in := #FC_NUMBER, out1 => "DB442_HOPPERS_ALARM_DECODING".GLOBAL_ALARMS_MACHINE.ALARM_DECODING)
      S_Coil( "DB442_HOPPERS_ALARM_DECODING".ALARMS_CENTRAL.IS_ALARMS )
   END_RUNG
   RUNG wire#w1
      { S7_GenerateENO := "TRUE" } Move(in := #FC_NUMBER, out1 => "DB441_POWDER_FEEDERS_ALARM_DECODING".GLOBAL_ALARMS_MACHINE.ALARM_DECODING)
      S_Coil( "DB441_POWDER_FEEDERS_ALARM_DECODING".ALARMS_CENTRAL.IS_ALARMS )
   END_RUNG
   // the same network as SCL:
   // ENO of a box is taken as its EN; it also drops when the box reports an error
   IF NOT (NOT "DB2100_GENERAL".EMERGENCY_STOP_ACTIVE_ALARM AND NOT "DB2100_GENERAL".ANY_AXIS_OR_CH_BYPASSED_ALARM AND NOT "DB2100_GENERAL".PROGRAMMING_ALARM AND NOT "DB2100_GENERAL".CHECK_NETWORK_LOGIC_ALARM) THEN
       "DB442_HOPPERS_ALARM_DECODING".GLOBAL_ALARMS_MACHINE.ALARM_DECODING := #FC_NUMBER;
       "DB442_HOPPERS_ALARM_DECODING".ALARMS_CENTRAL.IS_ALARMS := TRUE;
       "DB441_POWDER_FEEDERS_ALARM_DECODING".GLOBAL_ALARMS_MACHINE.ALARM_DECODING := #FC_NUMBER;
       "DB441_POWDER_FEEDERS_ALARM_DECODING".ALARMS_CENTRAL.IS_ALARMS := TRUE;
   END_IF;
END_REGION

REGION Network 9: CALL FC2103 ELECTRICAL CABINET
   RUNG wire#powerrail
      "FC2103_ELECTRICAL_CABINET"()
   END_RUNG
   // the same network as SCL:
   "FC2103_ELECTRICAL_CABINET"();
END_REGION

REGION Network 10: CALL FC2120 MPP ITC IPC
   RUNG wire#powerrail
      "FC2120_MPP_ITC_IPC"()
   END_RUNG
   // the same network as SCL:
   "FC2120_MPP_ITC_IPC"();
END_REGION

REGION Network 11: CALL FC2109 HOPPERS CONTROL ON
   RUNG wire#powerrail
      "FC2109_HOPPERS_CONTROL_ON"()
   END_RUNG
   // the same network as SCL:
   "FC2109_HOPPERS_CONTROL_ON"();
END_REGION

REGION Network 12: CALL FC2140 HOPPERS BUTTONS
   RUNG wire#powerrail
      "FC2140_HOPPERS_BUTTONS"()
   END_RUNG
   // the same network as SCL:
   "FC2140_HOPPERS_BUTTONS"();
END_REGION

REGION Network 13: CALL FC2141 HOPPERS LAMPS
   RUNG wire#powerrail
      "FC2141_HOPPERS_LAMPS"()
   END_RUNG
   // the same network as SCL:
   "FC2141_HOPPERS_LAMPS"();
END_REGION
END_FUNCTION

FUNCTION "FC2103_ELECTRICAL_CABINET" : Void   // FC2103, LAD
{ S7_Optimized_Access := 'FALSE' }
AUTHOR : ETXETAR
VERSION : 1.0
// stored: AutoNumber false, IsIECCheckEnabled false, SetENOAutomatically false, UDAEnableTagReadback false
   VAR CONSTANT
      FC_NUMBER : DInt := 2103;
   END_VAR
   VAR_TEMP   // added for the SCL form of the ladder/FBD networks
      _w1 : Bool;
   END_VAR
BEGIN

REGION Network 1: INPUTS
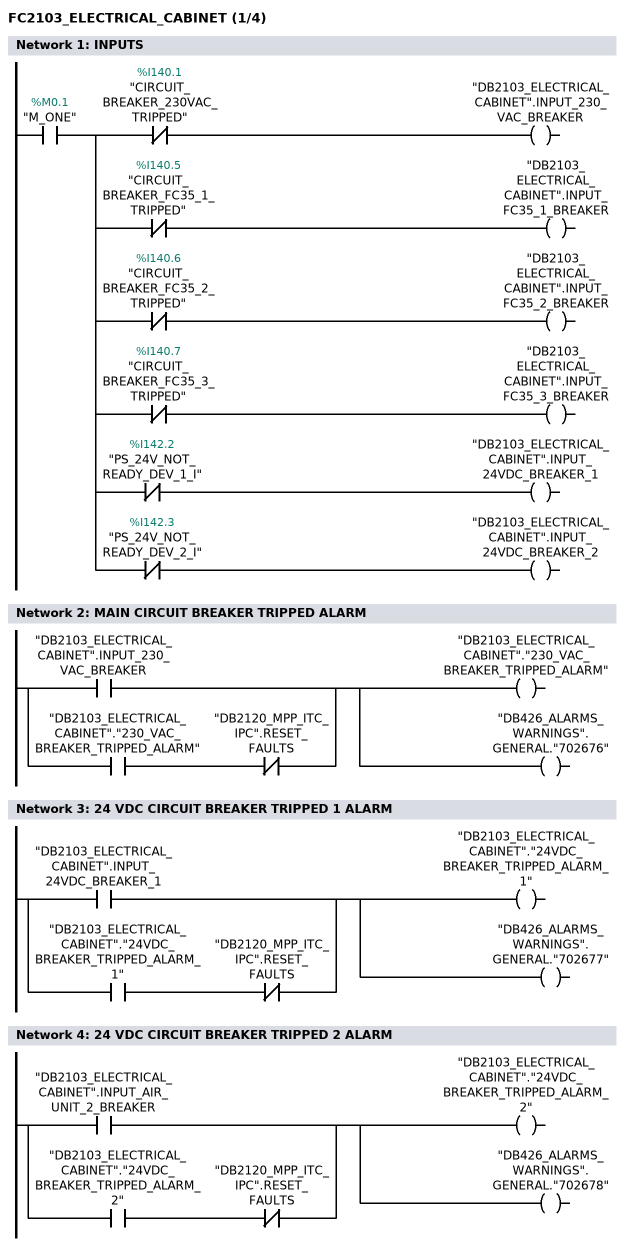
   RUNG wire#powerrail
      Contact( "M_ONE" )
      wire#w1
      I_Contact( "CIRCUIT_BREAKER_230VAC_TRIPPED" )
      Coil( "DB2103_ELECTRICAL_CABINET".INPUT_230_VAC_BREAKER )
   END_RUNG
   RUNG wire#w1
      I_Contact( "CIRCUIT_BREAKER_FC35_1_TRIPPED" )
      Coil( "DB2103_ELECTRICAL_CABINET".INPUT_FC35_1_BREAKER )
   END_RUNG
   RUNG wire#w1
      I_Contact( "CIRCUIT_BREAKER_FC35_2_TRIPPED" )
      Coil( "DB2103_ELECTRICAL_CABINET".INPUT_FC35_2_BREAKER )
   END_RUNG
   RUNG wire#w1
      I_Contact( "CIRCUIT_BREAKER_FC35_3_TRIPPED" )
      Coil( "DB2103_ELECTRICAL_CABINET".INPUT_FC35_3_BREAKER )
   END_RUNG
   RUNG wire#w1
      I_Contact( "PS_24V_NOT_READY_DEV_1_I" )
      Coil( "DB2103_ELECTRICAL_CABINET".INPUT_24VDC_BREAKER_1 )
   END_RUNG
   RUNG wire#w1
      I_Contact( "PS_24V_NOT_READY_DEV_2_I" )
      Coil( "DB2103_ELECTRICAL_CABINET".INPUT_24VDC_BREAKER_2 )
   END_RUNG
   // the same network as SCL:
   "DB2103_ELECTRICAL_CABINET".INPUT_230_VAC_BREAKER := "M_ONE" AND NOT "CIRCUIT_BREAKER_230VAC_TRIPPED";
   "DB2103_ELECTRICAL_CABINET".INPUT_FC35_1_BREAKER := "M_ONE" AND NOT "CIRCUIT_BREAKER_FC35_1_TRIPPED";
   "DB2103_ELECTRICAL_CABINET".INPUT_FC35_2_BREAKER := "M_ONE" AND NOT "CIRCUIT_BREAKER_FC35_2_TRIPPED";
   "DB2103_ELECTRICAL_CABINET".INPUT_FC35_3_BREAKER := "M_ONE" AND NOT "CIRCUIT_BREAKER_FC35_3_TRIPPED";
   "DB2103_ELECTRICAL_CABINET".INPUT_24VDC_BREAKER_1 := "M_ONE" AND NOT "PS_24V_NOT_READY_DEV_1_I";
   "DB2103_ELECTRICAL_CABINET".INPUT_24VDC_BREAKER_2 := "M_ONE" AND NOT "PS_24V_NOT_READY_DEV_2_I";
END_REGION

REGION Network 2: MAIN CIRCUIT BREAKER TRIPPED ALARM
   RUNG wire#powerrail
      Contact( "DB2103_ELECTRICAL_CABINET".INPUT_230_VAC_BREAKER )
      wire#w1
      Coil( "DB2103_ELECTRICAL_CABINET"."230_VAC_BREAKER_TRIPPED_ALARM" )
   END_RUNG
   RUNG wire#powerrail
      Contact( "DB2103_ELECTRICAL_CABINET"."230_VAC_BREAKER_TRIPPED_ALARM" )
      I_Contact( "DB2120_MPP_ITC_IPC".RESET_FAULTS )
   END_RUNG wire#w1
   RUNG wire#w1
      Coil( "DB426_ALARMS_WARNINGS".GENERAL."702676" )
   END_RUNG
   // the same network as SCL:
   "DB2103_ELECTRICAL_CABINET"."230_VAC_BREAKER_TRIPPED_ALARM" := "DB2103_ELECTRICAL_CABINET".INPUT_230_VAC_BREAKER OR ("DB2103_ELECTRICAL_CABINET"."230_VAC_BREAKER_TRIPPED_ALARM" AND NOT "DB2120_MPP_ITC_IPC".RESET_FAULTS);
   "DB426_ALARMS_WARNINGS".GENERAL."702676" := "DB2103_ELECTRICAL_CABINET"."230_VAC_BREAKER_TRIPPED_ALARM";
END_REGION

REGION Network 3: 24 VDC CIRCUIT BREAKER TRIPPED 1 ALARM
   RUNG wire#powerrail
      Contact( "DB2103_ELECTRICAL_CABINET".INPUT_24VDC_BREAKER_1 )
      wire#w1
      Coil( "DB2103_ELECTRICAL_CABINET"."24VDC_BREAKER_TRIPPED_ALARM_1" )
   END_RUNG
   RUNG wire#powerrail
      Contact( "DB2103_ELECTRICAL_CABINET"."24VDC_BREAKER_TRIPPED_ALARM_1" )
      I_Contact( "DB2120_MPP_ITC_IPC".RESET_FAULTS )
   END_RUNG wire#w1
   RUNG wire#w1
      Coil( "DB426_ALARMS_WARNINGS".GENERAL."702677" )
   END_RUNG
   // the same network as SCL:
   "DB2103_ELECTRICAL_CABINET"."24VDC_BREAKER_TRIPPED_ALARM_1" := "DB2103_ELECTRICAL_CABINET".INPUT_24VDC_BREAKER_1 OR ("DB2103_ELECTRICAL_CABINET"."24VDC_BREAKER_TRIPPED_ALARM_1" AND NOT "DB2120_MPP_ITC_IPC".RESET_FAULTS);
   "DB426_ALARMS_WARNINGS".GENERAL."702677" := "DB2103_ELECTRICAL_CABINET"."24VDC_BREAKER_TRIPPED_ALARM_1";
END_REGION

REGION Network 4: 24 VDC CIRCUIT BREAKER TRIPPED 2 ALARM
   RUNG wire#powerrail
      Contact( "DB2103_ELECTRICAL_CABINET".INPUT_AIR_UNIT_2_BREAKER )
      wire#w1
      Coil( "DB2103_ELECTRICAL_CABINET"."24VDC_BREAKER_TRIPPED_ALARM_2" )
   END_RUNG
   RUNG wire#powerrail
      Contact( "DB2103_ELECTRICAL_CABINET"."24VDC_BREAKER_TRIPPED_ALARM_2" )
      I_Contact( "DB2120_MPP_ITC_IPC".RESET_FAULTS )
   END_RUNG wire#w1
   RUNG wire#w1
      Coil( "DB426_ALARMS_WARNINGS".GENERAL."702678" )
   END_RUNG
   // the same network as SCL:
   "DB2103_ELECTRICAL_CABINET"."24VDC_BREAKER_TRIPPED_ALARM_2" := "DB2103_ELECTRICAL_CABINET".INPUT_AIR_UNIT_2_BREAKER OR ("DB2103_ELECTRICAL_CABINET"."24VDC_BREAKER_TRIPPED_ALARM_2" AND NOT "DB2120_MPP_ITC_IPC".RESET_FAULTS);
   "DB426_ALARMS_WARNINGS".GENERAL."702678" := "DB2103_ELECTRICAL_CABINET"."24VDC_BREAKER_TRIPPED_ALARM_2";
END_REGION

REGION Network 5: FC35_1 CIRCUIT BREAKER TRIPPED ALARM
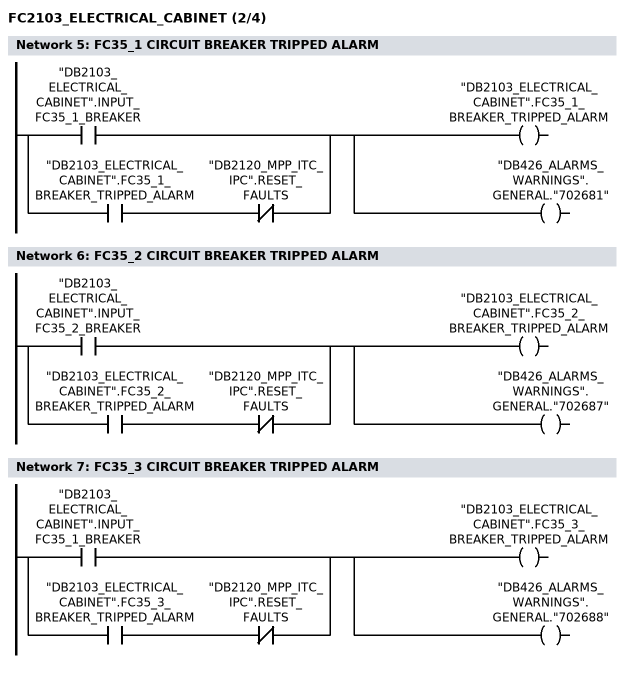
   RUNG wire#powerrail
      Contact( "DB2103_ELECTRICAL_CABINET".INPUT_FC35_1_BREAKER )
      wire#w1
      Coil( "DB2103_ELECTRICAL_CABINET".FC35_1_BREAKER_TRIPPED_ALARM )
   END_RUNG
   RUNG wire#powerrail
      Contact( "DB2103_ELECTRICAL_CABINET".FC35_1_BREAKER_TRIPPED_ALARM )
      I_Contact( "DB2120_MPP_ITC_IPC".RESET_FAULTS )
   END_RUNG wire#w1
   RUNG wire#w1
      Coil( "DB426_ALARMS_WARNINGS".GENERAL."702681" )
   END_RUNG
   // the same network as SCL:
   "DB2103_ELECTRICAL_CABINET".FC35_1_BREAKER_TRIPPED_ALARM := "DB2103_ELECTRICAL_CABINET".INPUT_FC35_1_BREAKER OR ("DB2103_ELECTRICAL_CABINET".FC35_1_BREAKER_TRIPPED_ALARM AND NOT "DB2120_MPP_ITC_IPC".RESET_FAULTS);
   "DB426_ALARMS_WARNINGS".GENERAL."702681" := "DB2103_ELECTRICAL_CABINET".FC35_1_BREAKER_TRIPPED_ALARM;
END_REGION

REGION Network 6: FC35_2 CIRCUIT BREAKER TRIPPED ALARM
   RUNG wire#powerrail
      Contact( "DB2103_ELECTRICAL_CABINET".INPUT_FC35_2_BREAKER )
      wire#w1
      Coil( "DB2103_ELECTRICAL_CABINET".FC35_2_BREAKER_TRIPPED_ALARM )
   END_RUNG
   RUNG wire#powerrail
      Contact( "DB2103_ELECTRICAL_CABINET".FC35_2_BREAKER_TRIPPED_ALARM )
      I_Contact( "DB2120_MPP_ITC_IPC".RESET_FAULTS )
   END_RUNG wire#w1
   RUNG wire#w1
      Coil( "DB426_ALARMS_WARNINGS".GENERAL."702687" )
   END_RUNG
   // the same network as SCL:
   "DB2103_ELECTRICAL_CABINET".FC35_2_BREAKER_TRIPPED_ALARM := "DB2103_ELECTRICAL_CABINET".INPUT_FC35_2_BREAKER OR ("DB2103_ELECTRICAL_CABINET".FC35_2_BREAKER_TRIPPED_ALARM AND NOT "DB2120_MPP_ITC_IPC".RESET_FAULTS);
   "DB426_ALARMS_WARNINGS".GENERAL."702687" := "DB2103_ELECTRICAL_CABINET".FC35_2_BREAKER_TRIPPED_ALARM;
END_REGION

REGION Network 7: FC35_3 CIRCUIT BREAKER TRIPPED ALARM
   RUNG wire#powerrail
      Contact( "DB2103_ELECTRICAL_CABINET".INPUT_FC35_1_BREAKER )
      wire#w1
      Coil( "DB2103_ELECTRICAL_CABINET".FC35_3_BREAKER_TRIPPED_ALARM )
   END_RUNG
   RUNG wire#powerrail
      Contact( "DB2103_ELECTRICAL_CABINET".FC35_3_BREAKER_TRIPPED_ALARM )
      I_Contact( "DB2120_MPP_ITC_IPC".RESET_FAULTS )
   END_RUNG wire#w1
   RUNG wire#w1
      Coil( "DB426_ALARMS_WARNINGS".GENERAL."702688" )
   END_RUNG
   // the same network as SCL:
   "DB2103_ELECTRICAL_CABINET".FC35_3_BREAKER_TRIPPED_ALARM := "DB2103_ELECTRICAL_CABINET".INPUT_FC35_1_BREAKER OR ("DB2103_ELECTRICAL_CABINET".FC35_3_BREAKER_TRIPPED_ALARM AND NOT "DB2120_MPP_ITC_IPC".RESET_FAULTS);
   "DB426_ALARMS_WARNINGS".GENERAL."702688" := "DB2103_ELECTRICAL_CABINET".FC35_3_BREAKER_TRIPPED_ALARM;
END_REGION

